C05461=1054.323,-117.646,435.270,170.401,28.686,155.440
C05462=1054.330,-117.397,435.261,170.403,28.687,155.440
C05463=1054.336,-117.147,435.251,170.405,28.688,155.440
C05464=1054.342,-116.897,435.242,170.407,28.688,155.440
C05465=1054.348,-116.647,435.232,170.409,28.689,155.440
C05466=1054.354,-116.397,435.222,170.410,28.689,155.440
C05467=1054.360,-116.148,435.213,170.412,28.689,155.440
C05468=1054.367,-115.898,435.203,170.415,28.691,155.440
C05469=1054.373,-115.648,435.194,170.417,28.691,155.440
C05470=1054.379,-115.364,435.183,170.419,28.692,155.440
C05471=1054.387,-115.080,435.172,170.422,28.692,155.440
C05472=1054.393,-114.795,435.162,170.424,28.693,155.440
C05473=1054.401,-114.511,435.150,170.427,28.694,155.439
C05474=1054.407,-114.261,435.141,170.428,28.694,155.439
C05475=1054.413,-114.011,435.131,170.430,28.695,155.439
C05476=1054.419,-113.762,435.122,170.432,28.696,155.439
C05477=1054.425,-113.512,435.113,170.434,28.696,155.439
C05478=1054.431,-113.263,435.103,170.436,28.697,155.439
C05479=1054.437,-113.013,435.092,170.439,28.698,155.439
C05480=1054.443,-112.763,435.083,170.441,28.698,155.439
C05481=1054.449,-112.514,435.073,170.443,28.699,155.439
C05482=1054.455,-112.264,435.063,170.445,28.699,155.439
C05483=1054.462,-112.014,435.054,170.446,28.700,155.439
C05484=1054.468,-111.764,435.044,170.448,28.701,155.439
C05485=1054.474,-111.514,435.035,170.450,28.702,155.439
C05486=1054.480,-111.265,435.025,170.453,28.702,155.439
C05487=1054.487,-111.015,435.015,170.455,28.703,155.439
C05488=1054.493,-110.766,435.005,170.457,28.704,155.439
C05489=1054.498,-110.515,434.995,170.459,28.704,155.439
C05490=1054.504,-110.266,434.986,170.461,28.705,155.439
C05491=1054.511,-110.016,434.976,170.462,28.706,155.439
C05492=1054.517,-109.766,434.966,170.465,28.706,155.438
C05493=1054.523,-109.517,434.956,170.467,28.707,155.438
C05494=1054.529,-109.267,434.947,170.469,28.708,155.438
C05495=1054.535,-109.017,434.937,170.471,28.708,155.438
C05496=1054.542,-108.768,434.927,170.473,28.709,155.438
C05497=1054.548,-108.518,434.917,170.475,28.710,155.438
C05498=1054.554,-108.268,434.907,170.477,28.711,155.438
C05499=1054.560,-108.018,434.897,170.479,28.711,155.438
C05500=1054.567,-107.768,434.888,170.481,28.712,155.438
C05501=1054.573,-107.519,434.877,170.483,28.713,155.438
C05502=1054.579,-107.269,434.868,170.485,28.713,155.438
C05503=1054.585,-107.019,434.858,170.487,28.714,155.438
C05504=1054.591,-106.769,434.848,170.489,28.715,155.438
C05505=1054.597,-106.520,434.838,170.491,28.716,155.438
C05506=1054.603,-106.270,434.828,170.494,28.716,155.438
C05507=1054.610,-106.020,434.819,170.495,28.717,155.438
C05508=1054.615,-105.771,434.808,170.497,28.719,155.438
C05509=1054.622,-105.521,434.798,170.499,28.719,155.438
C05510=1054.628,-105.271,434.789,170.501,28.720,155.438
C05511=1054.634,-105.022,434.778,170.503,28.720,155.438
C05512=1054.640,-104.772,434.768,170.505,28.721,155.438
C05513=1054.646,-104.521,434.758,170.508,28.722,155.438
C05514=1054.653,-104.272,434.748,170.509,28.723,155.438
C05515=1054.658,-104.022,434.738,170.511,28.724,155.438
C05516=1054.665,-103.773,434.727,170.513,28.725,155.438
C05517=1054.671,-103.523,434.718,170.515,28.726,155.438
C05518=1054.677,-103.273,434.708,170.517,28.726,155.438
C05519=1054.683,-103.024,434.697,170.519,28.727,155.438
C05520=1054.689,-102.774,434.688,170.522,28.728,155.438
C05521=1054.695,-102.525,434.678,170.523,28.729,155.438
C05522=1054.702,-102.274,434.667,170.525,28.730,155.438
C05523=1054.708,-102.025,434.657,170.527,28.731,155.438
C05524=1054.714,-101.775,434.647,170.529,28.731,155.438
C05525=1054.720,-101.525,434.637,170.531,28.732,155.438
C05526=1054.726,-101.276,434.627,170.533,28.733,155.438
C05527=1054.732,-101.026,434.617,170.536,28.734,155.437
C05528=1054.738,-100.777,434.606,170.537,28.735,155.438
C05529=1054.745,-100.526,434.596,170.539,28.736,155.438
C05530=1054.751,-100.277,434.586,170.541,28.737,155.437
C05531=1054.757,-100.027,434.576,170.543,28.738,155.437
C05532=1054.763,-99.778,434.566,170.545,28.739,155.438
C05533=1054.769,-99.527,434.555,170.547,28.739,155.437
C05534=1054.777,-99.242,434.544,170.550,28.740,155.437
C05535=1054.784,-98.956,434.532,170.551,28.741,155.437
C05536=1054.791,-98.670,434.521,170.554,28.743,155.437
C05537=1054.798,-98.385,434.508,170.556,28.744,155.437
C05538=1054.803,-98.135,434.498,170.558,28.744,155.437
C05539=1054.810,-97.886,434.488,170.560,28.745,155.437
C05540=1054.816,-97.636,434.478,170.563,28.746,155.437
C05541=1054.822,-97.386,434.467,170.564,28.747,155.437
C05542=1054.829,-97.137,434.457,170.566,28.748,155.437
C05543=1054.834,-96.887,434.447,170.568,28.749,155.437
C05544=1054.840,-96.637,434.436,170.570,28.750,155.437
C05545=1054.847,-96.388,434.425,170.572,28.751,155.437
C05546=1054.852,-96.138,434.415,170.574,28.752,155.438
C05547=1054.859,-95.888,434.405,170.575,28.753,155.438
C05548=1054.865,-95.638,434.394,170.578,28.754,155.438
C05549=1054.871,-95.389,434.384,170.580,28.755,155.438
C05550=1054.877,-95.139,434.373,170.582,28.756,155.438
C05551=1054.882,-94.890,434.362,170.584,28.757,155.438
C05552=1054.889,-94.639,434.352,170.586,28.758,155.438
C05553=1054.895,-94.390,434.342,170.587,28.759,155.438
C05554=1054.901,-94.140,434.331,170.589,28.760,155.438
C05555=1054.907,-93.890,434.321,170.591,28.761,155.438
C05556=1054.913,-93.641,434.310,170.594,28.763,155.438
C05557=1054.920,-93.391,434.300,170.596,28.763,155.438
C05558=1054.925,-93.141,434.289,170.598,28.764,155.438
C05559=1054.932,-92.892,434.279,170.600,28.765,155.438
C05560=1054.937,-92.642,434.268,170.601,28.766,155.438
C05561=1054.944,-92.392,434.257,170.603,28.767,155.438
C05562=1054.950,-92.143,434.247,170.605,28.768,155.438
C05563=1054.956,-91.893,434.237,170.607,28.769,155.438
C05564=1054.961,-91.643,434.226,170.610,28.771,155.438
C05565=1054.968,-91.393,434.215,170.611,28.772,155.438
C05566=1054.974,-91.144,434.204,170.613,28.773,155.438
C05567=1054.981,-90.895,434.194,170.615,28.774,155.438
C05568=1054.987,-90.644,434.183,170.617,28.775,155.438
C05569=1054.992,-90.394,434.173,170.619,28.776,155.438
C05570=1054.999,-90.145,434.162,170.621,28.777,155.438
C05571=1055.005,-89.895,434.151,170.622,28.778,155.438
C05572=1055.011,-89.645,434.140,170.624,28.780,155.438
C05573=1055.017,-89.396,434.130,170.627,28.781,155.438
C05574=1055.024,-89.146,434.119,170.629,28.782,155.438
C05575=1055.029,-88.896,434.108,170.631,28.783,155.438
C05576=1055.036,-88.647,434.098,170.633,28.784,155.438
C05577=1055.041,-88.397,434.087,170.634,28.785,155.438
C05578=1055.048,-88.147,434.076,170.636,28.786,155.438
C05579=1055.054,-87.898,434.066,170.638,28.787,155.438
C05580=1055.061,-87.648,434.055,170.640,28.788,155.438
C05581=1055.066,-87.398,434.044,170.643,28.789,155.438
C05582=1055.073,-87.149,434.033,170.645,28.790,155.438
C05583=1055.079,-86.899,434.022,170.646,28.791,155.439
C05584=1055.085,-86.649,434.011,170.648,28.792,155.439
C05585=1055.091,-86.400,434.001,170.650,28.794,155.439
C05586=1055.098,-86.150,433.990,170.652,28.795,155.439
C05587=1055.103,-85.901,433.979,170.654,28.796,155.439
C05588=1055.111,-85.651,433.968,170.656,28.797,155.439
C05589=1055.116,-85.401,433.957,170.657,28.798,155.439
C05590=1055.122,-85.152,433.946,170.660,28.799,155.439
C05591=1055.129,-84.902,433.936,170.662,28.800,155.439
C05592=1055.135,-84.652,433.925,170.664,28.801,155.439
C05593=1055.141,-84.402,433.914,170.666,28.803,155.439
C05594=1055.147,-84.153,433.903,170.667,28.804,155.439
C05595=1055.153,-83.903,433.892,170.669,28.805,155.439
C05596=1055.160,-83.653,433.881,170.671,28.806,155.439
C05597=1055.165,-83.404,433.870,170.673,28.807,155.439
C05598=1055.173,-83.120,433.858,170.676,28.808,155.439
C05599=1055.180,-82.837,433.846,170.678,28.810,155.439
C05600=1055.187,-82.553,433.833,170.680,28.811,155.439
C05601=1055.194,-82.270,433.821,170.682,28.812,155.439
C05602=1055.201,-82.020,433.810,170.684,28.814,155.439
C05603=1055.206,-81.771,433.799,170.686,28.815,155.440
C05604=1055.213,-81.521,433.788,170.688,28.816,155.440
C05605=1055.219,-81.271,433.777,170.689,28.817,155.440
C05606=1055.225,-81.021,433.766,170.691,28.818,155.440
C05607=1055.231,-80.772,433.755,170.694,28.820,155.440
C05608=1055.238,-80.522,433.745,170.696,28.821,155.440
C05609=1055.244,-80.273,433.733,170.698,28.822,155.440
C05610=1055.251,-80.023,433.722,170.700,28.823,155.440
C05611=1055.256,-79.773,433.711,170.701,28.825,155.440
C05612=1055.263,-79.523,433.700,170.703,28.826,155.440
C05613=1055.269,-79.274,433.689,170.705,28.827,155.440
C05614=1055.276,-79.024,433.678,170.707,28.828,155.440
C05615=1055.282,-78.775,433.666,170.709,28.829,155.440
C05616=1055.288,-78.525,433.655,170.710,28.830,155.440
C05617=1055.294,-78.275,433.644,170.713,28.832,155.440
C05618=1055.300,-78.025,433.633,170.715,28.833,155.440
C05619=1055.306,-77.776,433.622,170.717,28.835,155.441
C05620=1055.312,-77.526,433.610,170.719,28.836,155.441
C05621=1055.318,-77.276,433.599,170.720,28.837,155.441
C05622=1055.324,-77.026,433.588,170.722,28.839,155.441
C05623=1055.331,-76.777,433.577,170.724,28.840,155.441
C05624=1055.337,-76.527,433.565,170.726,28.841,155.441
C05625=1055.343,-76.278,433.554,170.728,28.842,155.441
C05626=1055.349,-76.027,433.543,170.730,28.843,155.441
C05627=1055.355,-75.779,433.532,170.731,28.845,155.441
C05628=1055.361,-75.528,433.520,170.734,28.846,155.441
C05629=1055.367,-75.279,433.509,170.736,28.848,155.441
C05630=1055.374,-75.029,433.498,170.738,28.849,155.441
C05631=1055.379,-74.780,433.487,170.739,28.851,155.441
C05632=1055.386,-74.530,433.475,170.741,28.852,155.442
C05633=1055.392,-74.281,433.464,170.743,28.853,155.442
C05634=1055.398,-74.031,433.453,170.745,28.854,155.442
C05635=1055.405,-73.780,433.441,170.747,28.856,155.442
C05636=1055.411,-73.532,433.430,170.749,28.857,155.442
C05637=1055.417,-73.281,433.418,170.750,28.859,155.442
C05638=1055.422,-73.032,433.406,170.752,28.860,155.442
C05639=1055.429,-72.782,433.395,170.754,28.861,155.442
C05640=1055.435,-72.533,433.383,170.757,28.863,155.442
C05641=1055.441,-72.283,433.372,170.758,28.864,155.442
C05642=1055.447,-72.033,433.361,170.760,28.866,155.442
C05643=1055.453,-71.784,433.349,170.762,28.867,155.443
C05644=1055.458,-71.534,433.338,170.764,28.868,155.443
C05645=1055.465,-71.284,433.326,170.766,28.870,155.443
C05646=1055.471,-71.035,433.315,170.767,28.872,155.443
C05647=1055.477,-70.785,433.303,170.769,28.873,155.443
C05648=1055.482,-70.536,433.292,170.771,28.874,155.443
C05649=1055.489,-70.286,433.280,170.773,28.876,155.443
C05650=1055.495,-70.036,433.268,170.775,28.877,155.443
C05651=1055.501,-69.787,433.256,170.776,28.879,155.443
C05652=1055.507,-69.536,433.245,170.778,28.880,155.444
C05653=1055.513,-69.288,433.233,170.780,28.881,155.444
C05654=1055.519,-69.037,433.222,170.783,28.883,155.444
C05655=1055.525,-68.788,433.210,170.784,28.885,155.444
C05656=1055.531,-68.538,433.199,170.786,28.886,155.444
C05657=1055.538,-68.288,433.187,170.788,28.887,155.444
C05658=1055.544,-68.040,433.175,170.790,28.889,155.444
C05659=1055.549,-67.789,433.163,170.792,28.891,155.444
C05660=1055.556,-67.540,433.151,170.793,28.892,155.444
C05661=1055.562,-67.290,433.141,170.795,28.893,155.445
C05662=1055.568,-67.009,433.127,170.797,28.895,155.445
C05663=1055.576,-66.728,433.114,170.800,28.897,155.445
C05664=1055.583,-66.446,433.100,170.801,28.898,155.445
C05665=1055.590,-66.165,433.087,170.803,28.900,155.445
C05666=1055.595,-65.915,433.076,170.805,28.902,155.445
C05667=1055.602,-65.666,433.064,170.807,28.903,155.445
C05668=1055.608,-65.416,433.052,170.809,28.904,155.445
C05669=1055.614,-65.167,433.041,170.810,28.906,155.446
C05670=1055.620,-64.917,433.028,170.813,28.908,155.446
C05671=1055.626,-64.667,433.016,170.815,28.909,155.446
C05672=1055.632,-64.418,433.006,170.817,28.911,155.446
C05673=1055.638,-64.168,432.993,170.819,28.912,155.446
C05674=1055.645,-63.918,432.981,170.820,28.914,155.446
C05675=1055.651,-63.669,432.970,170.822,28.915,155.446
C05676=1055.656,-63.419,432.958,170.824,28.916,155.446
C05677=1055.663,-63.169,432.946,170.826,28.918,155.447
C05678=1055.670,-62.920,432.934,170.827,28.920,155.447
C05679=1055.675,-62.670,432.922,170.829,28.921,155.447
C05680=1055.681,-62.421,432.910,170.831,28.922,155.447
C05681=1055.688,-62.171,432.898,170.833,28.924,155.447
C05682=1055.694,-61.921,432.886,170.835,28.926,155.447
C05683=1055.700,-61.672,432.875,170.836,28.927,155.447
C05684=1055.706,-61.422,432.863,170.838,28.929,155.448
C05685=1055.713,-61.172,432.851,170.840,28.930,155.448
C05686=1055.719,-60.923,432.838,170.842,28.932,155.448
C05687=1055.725,-60.674,432.827,170.844,28.933,155.448
C05688=1055.730,-60.423,432.815,170.845,28.935,155.448
C05689=1055.737,-60.174,432.803,170.848,28.937,155.448
C05690=1055.744,-59.924,432.791,170.850,28.938,155.448
C05691=1055.749,-59.675,432.779,170.852,28.939,155.448
C05692=1055.756,-59.425,432.767,170.853,28.941,155.448
C05693=1055.762,-59.175,432.756,170.855,28.943,155.449
C05694=1055.768,-58.925,432.743,170.857,28.944,155.449
C05695=1055.775,-58.676,432.731,170.859,28.946,155.449
C05696=1055.781,-58.427,432.720,170.861,28.947,155.449
C05697=1055.787,-58.177,432.707,170.862,28.949,155.449
C05698=1055.793,-57.927,432.695,170.864,28.950,155.449
C05699=1055.800,-57.678,432.683,170.866,28.952,155.449
C05700=1055.806,-57.428,432.671,170.868,28.953,155.450
C05701=1055.812,-57.179,432.659,170.869,28.955,155.450
C05702=1055.817,-56.928,432.647,170.871,28.957,155.450
C05703=1055.824,-56.679,432.635,170.873,28.958,155.450
C05704=1055.831,-56.429,432.623,170.875,28.960,155.450
C05705=1055.837,-56.179,432.611,170.877,28.961,155.450
C05706=1055.843,-55.930,432.599,170.878,28.962,155.450
C05707=1055.850,-55.680,432.587,170.880,28.964,155.450
C05708=1055.855,-55.431,432.575,170.882,28.966,155.451
C05709=1055.862,-55.182,432.563,170.884,28.967,155.451
C05710=1055.868,-54.932,432.550,170.885,28.969,155.451
C05711=1055.874,-54.682,432.538,170.887,28.971,155.451
C05712=1055.881,-54.433,432.526,170.890,28.972,155.451
C05713=1055.887,-54.183,432.514,170.892,28.974,155.451
C05714=1055.894,-53.933,432.502,170.894,28.976,155.451
C05715=1055.900,-53.683,432.489,170.895,28.977,155.452
C05716=1055.906,-53.434,432.477,170.897,28.979,155.452
C05717=1055.913,-53.184,432.465,170.899,28.981,155.452
C05718=1055.918,-52.935,432.453,170.901,28.982,155.452
C05719=1055.925,-52.685,432.441,170.902,28.983,155.452
C05720=1055.931,-52.435,432.428,170.904,28.985,155.452
C05721=1055.937,-52.186,432.416,170.906,28.986,155.452
C05722=1055.943,-51.936,432.404,170.908,28.988,155.453
C05723=1055.950,-51.686,432.392,170.910,28.990,155.453
C05724=1055.957,-51.437,432.379,170.911,28.991,155.453
C05725=1055.963,-51.188,432.367,170.913,28.993,155.453
C05726=1055.970,-50.907,432.353,170.915,28.995,155.453
C05727=1055.977,-50.628,432.339,170.918,28.997,155.453
C05728=1055.984,-50.347,432.325,170.919,28.999,155.454
C05729=1055.990,-50.067,432.312,170.921,29.000,155.454
C05730=1055.997,-49.818,432.299,170.923,29.002,155.454
C05731=1056.003,-49.569,432.286,170.925,29.004,155.454
C05732=1056.009,-49.319,432.274,170.926,29.006,155.454
C05733=1056.016,-49.069,432.262,170.928,29.007,155.454
C05734=1056.022,-48.819,432.249,170.930,29.009,155.455
C05735=1056.027,-48.571,432.236,170.932,29.011,155.455
C05736=1056.033,-48.321,432.224,170.933,29.013,155.455
C05737=1056.040,-48.071,432.212,170.935,29.014,155.455
C05738=1056.046,-47.821,432.199,170.937,29.016,155.455
C05739=1056.052,-47.571,432.187,170.939,29.018,155.455
C05740=1056.058,-47.322,432.174,170.941,29.019,155.456
C05741=1056.065,-47.073,432.162,170.942,29.021,155.456
C05742=1056.070,-46.823,432.149,170.944,29.023,155.456
C05743=1056.076,-46.573,432.137,170.946,29.025,155.456
C05744=1056.083,-46.324,432.123,170.948,29.026,155.456
C05745=1056.089,-46.074,432.111,170.949,29.028,155.456
C05746=1056.095,-45.824,432.099,170.951,29.030,155.457
C05747=1056.101,-45.575,432.085,170.953,29.032,155.457
C05748=1056.107,-45.325,432.073,170.955,29.033,155.457
C05749=1056.114,-45.075,432.061,170.956,29.035,155.457
C05750=1056.120,-44.826,432.048,170.958,29.037,155.457
C05751=1056.126,-44.576,432.035,170.960,29.039,155.458
C05752=1056.132,-44.326,432.023,170.962,29.041,155.458
C05753=1056.138,-44.077,432.009,170.963,29.042,155.458
C05754=1056.145,-43.828,431.997,170.965,29.044,155.458
C05755=1056.151,-43.578,431.985,170.967,29.046,155.458
C05756=1056.157,-43.328,431.972,170.969,29.048,155.458
C05757=1056.163,-43.078,431.959,170.970,29.049,155.459
C05758=1056.169,-42.829,431.946,170.972,29.051,155.459
C05759=1056.176,-42.580,431.934,170.974,29.053,155.459
C05760=1056.182,-42.330,431.921,170.976,29.055,155.459
C05761=1056.188,-42.081,431.908,170.978,29.056,155.459
C05762=1056.194,-41.831,431.895,170.979,29.058,155.460
C05763=1056.200,-41.581,431.883,170.981,29.060,155.460
C05764=1056.207,-41.332,431.870,170.983,29.062,155.460
C05765=1056.212,-41.082,431.858,170.984,29.064,155.460
C05766=1056.219,-40.833,431.844,170.986,29.066,155.460
C05767=1056.225,-40.583,431.832,170.988,29.067,155.461
C05768=1056.231,-40.334,431.819,170.990,29.069,155.461
C05769=1056.237,-40.084,431.807,170.992,29.071,155.461
C05770=1056.244,-39.835,431.793,170.993,29.073,155.461
C05771=1056.250,-39.584,431.780,170.995,29.074,155.461
C05772=1056.256,-39.335,431.767,170.997,29.076,155.462
C05773=1056.262,-39.085,431.755,170.999,29.078,155.462
C05774=1056.269,-38.836,431.741,171.000,29.080,155.462
C05775=1056.275,-38.586,431.729,171.002,29.082,155.462
C05776=1056.281,-38.337,431.716,171.004,29.084,155.462
C05777=1056.287,-38.087,431.703,171.006,29.085,155.462
C05778=1056.293,-37.837,431.690,171.007,29.087,155.463
C05779=1056.299,-37.587,431.677,171.009,29.089,155.463
C05780=1056.305,-37.338,431.664,171.011,29.091,155.463
C05781=1056.311,-37.089,431.651,171.013,29.093,155.463
C05782=1056.317,-36.839,431.638,171.014,29.095,155.463
C05783=1056.324,-36.589,431.624,171.016,29.097,155.464
C05784=1056.330,-36.339,431.612,171.018,29.099,155.464
C05785=1056.336,-36.090,431.599,171.020,29.100,155.464
C05786=1056.342,-35.841,431.585,171.021,29.103,155.464
C05787=1056.348,-35.591,431.573,171.023,29.104,155.464
C05788=1056.354,-35.342,431.559,171.025,29.106,155.465
C05789=1056.360,-35.092,431.547,171.026,29.108,155.465
C05790=1056.368,-34.812,431.531,171.028,29.110,155.465
C05791=1056.374,-34.533,431.517,171.030,29.112,155.465
C05792=1056.381,-34.253,431.503,171.032,29.114,155.466
C05793=1056.388,-33.974,431.487,171.033,29.116,155.466
C05794=1056.394,-33.724,431.475,171.035,29.119,155.466
C05795=1056.400,-33.475,431.461,171.037,29.120,155.466
C05796=1056.406,-33.226,431.448,171.039,29.122,155.467
C05797=1056.413,-32.975,431.435,171.040,29.124,155.467
C05798=1056.419,-32.726,431.422,171.042,29.126,155.467
C05799=1056.425,-32.477,431.409,171.044,29.128,155.467
C05800=1056.431,-32.227,431.395,171.046,29.130,155.467
C05801=1056.437,-31.977,431.383,171.047,29.132,155.468
C05802=1056.444,-31.728,431.369,171.049,29.134,155.468
C05803=1056.450,-31.478,431.356,171.051,29.135,155.468
C05804=1056.457,-31.229,431.343,171.053,29.138,155.468
C05805=1056.462,-30.979,431.329,171.054,29.139,155.468
C05806=1056.468,-30.729,431.316,171.056,29.142,155.469
C05807=1056.474,-30.480,431.303,171.058,29.143,155.469
C05808=1056.481,-30.230,431.289,171.060,29.145,155.469
C05809=1056.487,-29.980,431.277,171.061,29.147,155.469
C05810=1056.493,-29.731,431.263,171.063,29.149,155.470
C05811=1056.499,-29.482,431.250,171.064,29.151,155.470
C05812=1056.506,-29.232,431.236,171.066,29.153,155.470
C05813=1056.512,-28.983,431.223,171.068,29.154,155.470
C05814=1056.518,-28.733,431.209,171.069,29.157,155.470
C05815=1056.524,-28.483,431.197,171.071,29.158,155.471
C05816=1056.530,-28.234,431.183,171.073,29.160,155.471
C05817=1056.537,-27.984,431.170,171.075,29.162,155.471
C05818=1056.543,-27.735,431.157,171.076,29.164,155.471
C05819=1056.549,-27.485,431.143,171.078,29.166,155.472
C05820=1056.556,-27.235,431.130,171.080,29.168,155.472
C05821=1056.562,-26.986,431.116,171.081,29.170,155.472
C05822=1056.568,-26.737,431.103,171.083,29.172,155.472
C05823=1056.574,-26.487,431.089,171.085,29.174,155.472
C05824=1056.581,-26.237,431.076,171.087,29.176,155.473
C05825=1056.586,-25.987,431.062,171.088,29.178,155.473
C05826=1056.592,-25.738,431.049,171.090,29.180,155.473
C05827=1056.598,-25.489,431.036,171.092,29.182,155.473
C05828=1056.604,-25.238,431.022,171.093,29.184,155.474
C05829=1056.611,-24.989,431.008,171.094,29.186,155.474
C05830=1056.617,-24.740,430.995,171.096,29.188,155.474
C05831=1056.622,-24.490,430.981,171.098,29.190,155.474
C05832=1056.629,-24.240,430.968,171.100,29.192,155.474
C05833=1056.635,-23.991,430.954,171.101,29.194,155.475
C05834=1056.641,-23.741,430.941,171.103,29.196,155.475
C05835=1056.647,-23.492,430.927,171.105,29.198,155.475
C05836=1056.653,-23.242,430.913,171.107,29.200,155.475
C05837=1056.659,-22.993,430.900,171.108,29.202,155.476
C05838=1056.666,-22.744,430.886,171.110,29.205,155.476
C05839=1056.672,-22.494,430.872,171.112,29.206,155.476
C05840=1056.678,-22.244,430.858,171.114,29.208,155.476
C05841=1056.684,-21.995,430.845,171.115,29.211,155.477
C05842=1056.690,-21.745,430.831,171.116,29.212,155.477
C05843=1056.697,-21.496,430.818,171.118,29.214,155.477
C05844=1056.702,-21.246,430.804,171.120,29.216,155.477
C05845=1056.709,-20.996,430.790,171.121,29.219,155.478
C05846=1056.715,-20.747,430.777,171.123,29.220,155.478
C05847=1056.721,-20.497,430.763,171.125,29.222,155.478
C05848=1056.727,-20.247,430.749,171.126,29.225,155.478
C05849=1056.733,-19.998,430.735,171.128,29.227,155.479
C05850=1056.739,-19.749,430.721,171.130,29.228,155.479
C05851=1056.746,-19.499,430.708,171.132,29.231,155.479
C05852=1056.752,-19.249,430.694,171.133,29.233,155.479
C05853=1056.758,-19.000,430.681,171.135,29.235,155.480
C05854=1056.765,-18.720,430.664,171.137,29.237,155.480
C05855=1056.772,-18.440,430.649,171.139,29.239,155.480
C05856=1056.779,-18.159,430.634,171.140,29.242,155.480
C05857=1056.786,-17.879,430.618,171.142,29.244,155.481
C05858=1056.792,-17.630,430.604,171.144,29.246,155.481
C05859=1056.798,-17.380,430.591,171.146,29.248,155.481
C05860=1056.804,-17.130,430.577,171.147,29.250,155.481
C05861=1056.811,-16.881,430.563,171.149,29.252,155.482
C05862=1056.818,-16.631,430.549,171.151,29.254,155.482
C05863=1056.823,-16.382,430.535,171.153,29.256,155.482
C05864=1056.829,-16.133,430.522,171.153,29.258,155.482
C05865=1056.836,-15.883,430.507,171.155,29.260,155.483
C05866=1056.842,-15.634,430.494,171.157,29.262,155.483
C05867=1056.848,-15.383,430.480,171.158,29.264,155.483
C05868=1056.854,-15.134,430.466,171.160,29.266,155.483
C05869=1056.861,-14.884,430.451,171.162,29.268,155.484
C05870=1056.867,-14.635,430.438,171.164,29.270,155.484
C05871=1056.872,-14.386,430.424,171.165,29.273,155.484
C05872=1056.879,-14.136,430.409,171.167,29.275,155.484
C05873=1056.885,-13.887,430.396,171.169,29.277,155.485
C05874=1056.891,-13.636,430.382,171.170,29.279,155.485
C05875=1056.897,-13.388,430.368,171.171,29.281,155.485
C05876=1056.903,-13.138,430.354,171.173,29.283,155.486
C05877=1056.909,-12.889,430.339,171.175,29.285,155.486
C05878=1056.916,-12.639,430.326,171.177,29.287,155.486
C05879=1056.922,-12.389,430.312,171.178,29.289,155.486
C05880=1056.927,-12.140,430.297,171.180,29.292,155.487
C05881=1056.934,-11.890,430.283,171.182,29.294,155.487
C05882=1056.940,-11.641,430.269,171.184,29.296,155.487
C05883=1056.946,-11.391,430.254,171.184,29.298,155.487
C05884=1056.952,-11.142,430.241,171.186,29.300,155.488
C05885=1056.958,-10.893,430.227,171.188,29.302,155.488
C05886=1056.964,-10.642,430.212,171.189,29.305,155.488
C05887=1056.971,-10.394,430.198,171.191,29.307,155.488
C05888=1056.977,-10.143,430.184,171.193,29.309,155.489
C05889=1056.983,-9.894,430.170,171.195,29.311,155.489
C05890=1056.989,-9.644,430.156,171.196,29.313,155.489
C05891=1056.995,-9.396,430.141,171.197,29.315,155.489
C05892=1057.001,-9.145,430.127,171.199,29.317,155.490
C05893=1057.008,-8.897,430.113,171.201,29.319,155.490
C05894=1057.014,-8.646,430.099,171.202,29.321,155.490
C05895=1057.020,-8.397,430.084,171.204,29.324,155.491
C05896=1057.026,-8.147,430.070,171.206,29.326,155.491
C05897=1057.032,-7.898,430.056,171.208,29.328,155.491
C05898=1057.038,-7.648,430.042,171.209,29.330,155.491
C05899=1057.045,-7.399,430.027,171.210,29.332,155.492
C05900=1057.051,-7.149,430.014,171.212,29.334,155.492
C05901=1057.057,-6.900,429.999,171.214,29.337,155.492
C05902=1057.063,-6.650,429.985,171.215,29.339,155.493
C05903=1057.070,-6.401,429.971,171.217,29.341,155.493
C05904=1057.076,-6.152,429.956,171.219,29.343,155.493
C05905=1057.082,-5.901,429.942,171.220,29.345,155.493
C05906=1057.087,-5.652,429.927,171.222,29.348,155.494
C05907=1057.094,-5.403,429.914,171.223,29.350,155.494
C05908=1057.101,-5.153,429.899,171.225,29.352,155.494
C05909=1057.106,-4.904,429.884,171.226,29.353,155.494
C05910=1057.113,-4.654,429.870,171.228,29.356,155.495
C05911=1057.119,-4.405,429.856,171.230,29.358,155.495
C05912=1057.125,-4.155,429.841,171.232,29.360,155.495
C05913=1057.131,-3.905,429.827,171.233,29.362,155.495
C05914=1057.138,-3.656,429.813,171.235,29.364,155.496
C05915=1057.144,-3.407,429.798,171.236,29.366,155.496
C05916=1057.150,-3.157,429.784,171.238,29.368,155.496
C05917=1057.156,-2.908,429.769,171.239,29.371,155.497
C05918=1057.163,-2.625,429.752,171.241,29.373,155.497
C05919=1057.169,-2.344,429.736,171.243,29.376,155.497
C05920=1057.177,-2.062,429.720,171.244,29.378,155.498
C05921=1057.184,-1.780,429.703,171.246,29.381,155.498
C05922=1057.189,-1.531,429.688,171.248,29.383,155.498
C05923=1057.196,-1.281,429.674,171.250,29.386,155.499
C05924=1057.201,-1.032,429.660,171.251,29.388,155.499
C05925=1057.208,-0.782,429.645,171.253,29.390,155.499
C05926=1057.214,-0.532,429.630,171.255,29.392,155.499
C05927=1057.220,-0.284,429.615,171.256,29.395,155.500
C05928=1057.226,-0.033,429.601,171.257,29.397,155.500
C05929=1057.232,0.216,429.586,171.259,29.399,155.500
C05930=1057.238,0.465,429.571,171.261,29.401,155.501
C05931=1057.244,0.715,429.556,171.262,29.404,155.501
C05932=1057.250,0.964,429.542,171.264,29.406,155.501
C05933=1057.257,1.214,429.527,171.266,29.408,155.501
C05934=1057.262,1.463,429.513,171.267,29.410,155.502
C05935=1057.268,1.713,429.498,171.268,29.413,155.502
C05936=1057.274,1.963,429.483,171.270,29.415,155.502
C05937=1057.280,2.212,429.468,171.272,29.417,155.503
C05938=1057.286,2.461,429.453,171.274,29.419,155.503
C05939=1057.293,2.711,429.438,171.275,29.421,155.503
C05940=1057.298,2.960,429.424,171.276,29.423,155.504
C05941=1057.305,3.210,429.409,171.278,29.426,155.504
C05942=1057.311,3.460,429.394,171.279,29.428,155.504
C05943=1057.317,3.709,429.380,171.281,29.431,155.504
C05944=1057.323,3.959,429.365,171.283,29.433,155.505
C05945=1057.329,4.208,429.350,171.285,29.435,155.505
C05946=1057.335,4.457,429.335,171.285,29.437,155.505
C05947=1057.342,4.707,429.320,171.287,29.440,155.506
C05948=1057.348,4.957,429.305,171.289,29.442,155.506
C05949=1057.354,5.205,429.291,171.291,29.444,155.506
C05950=1057.360,5.455,429.276,171.292,29.446,155.507
C05951=1057.366,5.705,429.261,171.294,29.448,155.507
C05952=1057.372,5.954,429.246,171.295,29.450,155.507
C05953=1057.378,6.204,429.231,171.296,29.453,155.508
C05954=1057.384,6.453,429.216,171.298,29.455,155.508
C05955=1057.391,6.703,429.201,171.300,29.458,155.508
C05956=1057.396,6.952,429.186,171.302,29.460,155.508
C05957=1057.403,7.202,429.171,171.303,29.462,155.509
C05958=1057.409,7.451,429.156,171.304,29.464,155.509
C05959=1057.415,7.700,429.142,171.306,29.467,155.509
C05960=1057.421,7.950,429.127,171.308,29.469,155.510
C05961=1057.428,8.200,429.112,171.309,29.471,155.510
C05962=1057.434,8.449,429.097,171.311,29.473,155.510
C05963=1057.440,8.698,429.082,171.313,29.475,155.510
C05964=1057.446,8.948,429.067,171.314,29.477,155.511
C05965=1057.452,9.198,429.052,171.315,29.480,155.511
C05966=1057.459,9.447,429.036,171.317,29.482,155.511
C05967=1057.465,9.696,429.021,171.319,29.485,155.512
C05968=1057.471,9.945,429.007,171.321,29.487,155.512
C05969=1057.477,10.195,428.992,171.322,29.489,155.512
C05970=1057.484,10.445,428.977,171.323,29.491,155.513
C05971=1057.490,10.694,428.962,171.325,29.494,155.513
C05972=1057.495,10.944,428.947,171.326,29.496,155.513
C05973=1057.501,11.193,428.932,171.328,29.498,155.513
C05974=1057.508,11.442,428.916,171.330,29.500,155.514
C05975=1057.514,11.692,428.901,171.332,29.502,155.514
C05976=1057.521,11.942,428.886,171.332,29.504,155.514
C05977=1057.527,12.191,428.871,171.334,29.507,155.515
C05978=1057.533,12.440,428.857,171.336,29.509,155.515
C05979=1057.539,12.690,428.842,171.338,29.512,155.515
C05980=1057.545,12.939,428.826,171.339,29.514,155.516
C05981=1057.552,13.189,428.811,171.340,29.516,155.516
C05982=1057.559,13.472,428.794,171.342,29.518,155.516
C05983=1057.566,13.756,428.776,171.344,29.521,155.517
C05984=1057.573,14.041,428.759,171.346,29.524,155.517
C05985=1057.580,14.324,428.742,171.348,29.526,155.517
C05986=1057.587,14.573,428.727,171.350,29.529,155.518
C05987=1057.592,14.823,428.711,171.350,29.531,155.518
C05988=1057.599,15.073,428.696,171.352,29.533,155.518
C05989=1057.604,15.322,428.681,171.354,29.536,155.519
C05990=1057.610,15.571,428.666,171.356,29.538,155.519
C05991=1057.617,15.821,428.651,171.357,29.540,155.519
C05992=1057.623,16.070,428.634,171.358,29.542,155.519
C05993=1057.629,16.320,428.619,171.360,29.545,155.520
C05994=1057.636,16.570,428.604,171.361,29.547,155.520
C05995=1057.641,16.818,428.589,171.363,29.550,155.520
C05996=1057.647,17.068,428.574,171.365,29.552,155.521
C05997=1057.653,17.318,428.558,171.366,29.554,155.521
C05998=1057.660,17.567,428.542,171.367,29.556,155.521
C05999=1057.666,17.817,428.527,171.369,29.559,155.522
C06000=1057.672,18.067,428.512,171.371,29.561,155.522
C06001=1057.678,18.316,428.496,171.373,29.564,155.522
C06002=1057.684,18.565,428.482,171.373,29.566,155.523
C06003=1057.690,18.814,428.465,171.375,29.568,155.523
C06004=1057.697,19.064,428.451,171.377,29.571,155.523
C06005=1057.702,19.313,428.435,171.379,29.573,155.524
C06006=1057.709,19.563,428.419,171.380,29.575,155.524
C06007=1057.715,19.812,428.404,171.381,29.577,155.524
C06008=1057.721,20.062,428.388,171.383,29.580,155.525
C06009=1057.728,20.311,428.373,171.385,29.582,155.525
C06010=1057.734,20.561,428.357,171.386,29.585,155.525
C06011=1057.739,20.809,428.342,171.388,29.587,155.526
C06012=1057.745,21.059,428.326,171.389,29.589,155.526
C06013=1057.752,21.308,428.311,171.390,29.592,155.526
C06014=1057.758,21.558,428.295,171.392,29.594,155.527
C06015=1057.764,21.807,428.280,171.394,29.596,155.527
C06016=1057.770,22.057,428.264,171.395,29.598,155.527
C06017=1057.776,22.307,428.249,171.396,29.601,155.527
C06018=1057.782,22.556,428.232,171.398,29.603,155.528
C06019=1057.789,22.806,428.218,171.400,29.606,155.528
C06020=1057.795,23.055,428.201,171.402,29.608,155.528
C06021=1057.800,23.305,428.186,171.402,29.610,155.529
C06022=1057.807,23.554,428.170,171.404,29.612,155.529
C06023=1057.812,23.803,428.155,171.406,29.615,155.530
C06024=1057.819,24.052,428.139,171.408,29.617,155.530
C06025=1057.825,24.302,428.123,171.409,29.620,155.530
C06026=1057.831,24.551,428.108,171.410,29.622,155.531
C06027=1057.837,24.801,428.092,171.412,29.624,155.531
C06028=1057.843,25.050,428.077,171.413,29.626,155.531
C06029=1057.849,25.300,428.061,171.415,29.629,155.531
C06030=1057.856,25.549,428.045,171.416,29.631,155.532
C06031=1057.862,25.799,428.029,171.418,29.634,155.532
C06032=1057.868,26.048,428.013,171.419,29.636,155.532
C06033=1057.874,26.298,427.998,171.421,29.638,155.533
C06034=1057.880,26.547,427.982,171.423,29.641,155.533
C06035=1057.887,26.796,427.966,171.424,29.643,155.533
C06036=1057.892,27.046,427.951,171.425,29.646,155.534
C06037=1057.898,27.295,427.934,171.427,29.648,155.534
C06038=1057.905,27.544,427.919,171.429,29.650,155.534
C06039=1057.910,27.794,427.903,171.431,29.653,155.535
C06040=1057.917,28.043,427.888,171.431,29.655,155.535
C06041=1057.923,28.293,427.871,171.433,29.658,155.535
C06042=1057.929,28.542,427.855,171.435,29.660,155.536
C06043=1057.935,28.792,427.840,171.437,29.662,155.536
C06044=1057.941,29.041,427.824,171.437,29.665,155.536
C06045=1057.947,29.290,427.808,171.439,29.667,155.537
C06046=1057.954,29.576,427.789,171.441,29.669,155.537
C06047=1057.962,29.861,427.772,171.442,29.672,155.538
C06048=1057.968,30.145,427.753,171.444,29.675,155.538
C06049=1057.975,30.431,427.735,171.446,29.678,155.538
C06050=1057.981,30.680,427.718,171.447,29.681,155.539
C06051=1057.987,30.930,427.704,171.449,29.683,155.539
C06052=1057.993,31.179,427.687,171.451,29.685,155.539
C06053=1057.999,31.429,427.671,171.452,29.687,155.540
C06054=1058.005,31.678,427.655,171.453,29.690,155.540
C06055=1058.012,31.927,427.639,171.455,29.692,155.540
C06056=1058.018,32.176,427.623,171.457,29.695,155.541
C06057=1058.024,32.427,427.607,171.458,29.697,155.541
C06058=1058.030,32.676,427.591,171.459,29.700,155.541
C06059=1058.036,32.926,427.574,171.461,29.702,155.542
C06060=1058.043,33.175,427.559,171.463,29.704,155.542
C06061=1058.049,33.424,427.543,171.465,29.707,155.542
C06062=1058.055,33.673,427.526,171.465,29.709,155.543
C06063=1058.061,33.923,427.510,171.467,29.712,155.543
C06064=1058.066,34.172,427.494,171.469,29.714,155.543
C06065=1058.073,34.422,427.479,171.471,29.717,155.544
C06066=1058.079,34.671,427.463,171.471,29.719,155.544
C06067=1058.085,34.920,427.446,171.473,29.721,155.544
C06068=1058.091,35.170,427.430,171.475,29.723,155.545
C06069=1058.097,35.419,427.414,171.476,29.726,155.545
C06070=1058.104,35.669,427.398,171.478,29.728,155.545
C06071=1058.110,35.918,427.381,171.479,29.731,155.546
C06072=1058.116,36.168,427.365,171.481,29.733,155.546
C06073=1058.122,36.417,427.349,171.482,29.736,155.547
C06074=1058.128,36.666,427.333,171.484,29.738,155.547
C06075=1058.134,36.915,427.317,171.485,29.740,155.547
C06076=1058.140,37.165,427.301,171.487,29.743,155.548
C06077=1058.146,37.414,427.285,171.488,29.745,155.548
C06078=1058.153,37.664,427.268,171.490,29.748,155.548
C06079=1058.159,37.913,427.252,171.491,29.750,155.549
C06080=1058.165,38.163,427.235,171.493,29.752,155.549
C06081=1058.171,38.412,427.219,171.494,29.755,155.549
C06082=1058.177,38.661,427.203,171.496,29.757,155.550
C06083=1058.183,38.911,427.187,171.497,29.760,155.550
C06084=1058.189,39.160,427.170,171.499,29.762,155.550
C06085=1058.195,39.409,427.154,171.500,29.765,155.551
C06086=1058.201,39.660,427.138,171.502,29.767,155.551
C06087=1058.207,39.908,427.121,171.504,29.770,155.551
C06088=1058.213,40.158,427.104,171.505,29.772,155.552
C06089=1058.219,40.407,427.088,171.506,29.774,155.552
C06090=1058.225,40.656,427.072,171.508,29.777,155.552
C06091=1058.231,40.906,427.056,171.510,29.779,155.553
C06092=1058.237,41.155,427.039,171.510,29.782,155.553
C06093=1058.244,41.405,427.023,171.512,29.784,155.553
C06094=1058.250,41.654,427.006,171.514,29.787,155.554
C06095=1058.256,41.903,426.989,171.516,29.789,155.554
C06096=1058.262,42.152,426.973,171.516,29.792,155.555
C06097=1058.268,42.402,426.957,171.518,29.794,155.555
C06098=1058.274,42.651,426.941,171.520,29.796,155.555
C06099=1058.280,42.901,426.924,171.522,29.799,155.556
C06100=1058.286,43.151,426.908,171.522,29.801,155.556
C06101=1058.293,43.399,426.891,171.524,29.804,155.556
C06102=1058.299,43.693,426.871,171.526,29.807,155.557
C06103=1058.306,43.986,426.852,171.528,29.809,155.557
C06104=1058.313,44.279,426.833,171.529,29.813,155.558
C06105=1058.320,44.572,426.813,171.531,29.815,155.558
C06106=1058.326,44.817,426.796,171.533,29.818,155.558
C06107=1058.332,45.062,426.780,171.534,29.820,155.559
C06108=1058.337,45.308,426.764,171.536,29.823,155.559
C06109=1058.344,45.554,426.747,171.537,29.825,155.559
C06110=1058.349,45.799,426.731,171.539,29.828,155.560
C06111=1058.355,46.044,426.714,171.540,29.831,155.560
C06112=1058.361,46.289,426.697,171.541,29.833,155.561
C06113=1058.366,46.535,426.681,171.543,29.835,155.561
C06114=1058.372,46.784,426.665,171.545,29.838,155.561
C06115=1058.379,47.034,426.648,171.546,29.840,155.562
C06116=1058.384,47.283,426.631,171.547,29.843,155.562
C06117=1058.391,47.532,426.614,171.549,29.846,155.562
C06118=1058.397,47.782,426.598,171.551,29.848,155.563
C06119=1058.403,48.032,426.581,171.552,29.850,155.563
C06120=1058.409,48.281,426.563,171.553,29.853,155.564
C06121=1058.415,48.530,426.547,171.555,29.855,155.564
C06122=1058.421,48.779,426.531,171.556,29.858,155.564
C06123=1058.426,49.028,426.513,171.558,29.861,155.565
C06124=1058.433,49.278,426.497,171.559,29.863,155.565
C06125=1058.439,49.527,426.480,171.561,29.865,155.565
C06126=1058.445,49.776,426.464,171.562,29.868,155.566
C06127=1058.450,50.026,426.447,171.564,29.870,155.566
C06128=1058.457,50.276,426.429,171.565,29.873,155.566
C06129=1058.463,50.525,426.413,171.567,29.875,155.567
C06130=1058.469,50.774,426.395,171.568,29.878,155.567
C06131=1058.475,51.024,426.379,171.570,29.880,155.567
C06132=1058.481,51.273,426.362,171.571,29.882,155.568
C06133=1058.487,51.522,426.345,171.573,29.885,155.568
C06134=1058.493,51.771,426.328,171.574,29.888,155.569
C06135=1058.499,52.021,426.311,171.576,29.890,155.569
C06136=1058.505,52.270,426.294,171.577,29.893,155.569
C06137=1058.511,52.520,426.278,171.579,29.895,155.570
C06138=1058.518,52.769,426.260,171.580,29.897,155.570
C06139=1058.523,53.019,426.243,171.582,29.900,155.570
C06140=1058.529,53.267,426.226,171.583,29.903,155.571
C06141=1058.536,53.517,426.210,171.585,29.905,155.571
C06142=1058.541,53.766,426.192,171.586,29.908,155.571
C06143=1058.547,54.016,426.176,171.588,29.910,155.572
C06144=1058.554,54.265,426.159,171.589,29.912,155.572
C06145=1058.559,54.515,426.142,171.591,29.915,155.573
C06146=1058.565,54.764,426.125,171.592,29.917,155.573
C06147=1058.572,55.013,426.108,171.594,29.920,155.573
C06148=1058.578,55.263,426.091,171.595,29.923,155.574
C06149=1058.584,55.511,426.074,171.597,29.925,155.574
C06150=1058.590,55.762,426.057,171.598,29.927,155.574
C06151=1058.596,56.011,426.040,171.600,29.930,155.575
C06152=1058.602,56.259,426.023,171.601,29.932,155.575
C06153=1058.608,56.510,426.005,171.603,29.935,155.576
C06154=1058.614,56.758,425.988,171.604,29.937,155.576
C06155=1058.621,57.008,425.971,171.606,29.940,155.576
C06156=1058.626,57.257,425.954,171.607,29.942,155.577
C06157=1058.633,57.506,425.937,171.609,29.944,155.577
C06158=1058.639,57.756,425.921,171.610,29.947,155.577
C06159=1058.645,58.005,425.903,171.612,29.950,155.578
C06160=1058.651,58.255,425.886,171.613,29.952,155.578
C06161=1058.657,58.504,425.868,171.614,29.955,155.578
C06162=1058.663,58.753,425.852,171.616,29.957,155.579
C06163=1058.670,59.003,425.834,171.618,29.959,155.579
C06164=1058.675,59.252,425.817,171.619,29.962,155.580
C06165=1058.682,59.502,425.800,171.621,29.964,155.580
C06166=1058.687,59.751,425.783,171.622,29.967,155.580
C06167=1058.694,60.000,425.765,171.624,29.969,155.580
C06168=1058.700,60.249,425.748,171.625,29.972,155.581
C06169=1058.706,60.499,425.731,171.626,29.974,155.581
C06170=1058.713,60.748,425.714,171.628,29.976,155.582
C06171=1058.718,60.997,425.697,171.630,29.979,155.582
C06172=1058.725,61.246,425.679,171.631,29.981,155.582
C06173=1058.731,61.496,425.663,171.633,29.984,155.583
C06174=1058.738,61.781,425.642,171.634,29.987,155.583
C06175=1058.745,62.066,425.623,171.636,29.989,155.584
C06176=1058.752,62.351,425.603,171.638,29.992,155.584
C06177=1058.759,62.635,425.583,171.639,29.995,155.584
C06178=1058.766,62.885,425.567,171.641,29.998,155.585
C06179=1058.771,63.134,425.549,171.643,30.000,155.585
C06180=1058.778,63.383,425.532,171.644,30.002,155.585
C06181=1058.784,63.632,425.514,171.645,30.005,155.586
C06182=1058.791,63.882,425.497,171.647,30.007,155.586
C06183=1058.796,64.131,425.479,171.649,30.010,155.587
C06184=1058.803,64.380,425.462,171.651,30.012,155.587
C06185=1058.808,64.630,425.445,171.651,30.015,155.587
C06186=1058.815,64.879,425.428,171.653,30.017,155.588
C06187=1058.821,65.128,425.410,171.655,30.020,155.588
C06188=1058.827,65.378,425.392,171.656,30.022,155.588
C06189=1058.833,65.627,425.375,171.657,30.025,155.589
C06190=1058.839,65.876,425.358,171.659,30.027,155.589
C06191=1058.845,66.126,425.340,171.661,30.030,155.589
C06192=1058.851,66.374,425.323,171.662,30.032,155.590
C06193=1058.857,66.624,425.305,171.663,30.035,155.590
C06194=1058.863,66.873,425.287,171.665,30.038,155.591
C06195=1058.869,67.123,425.270,171.667,30.040,155.591
C06196=1058.876,67.372,425.252,171.668,30.042,155.591
C06197=1058.881,67.621,425.235,171.669,30.045,155.592
C06198=1058.887,67.871,425.217,171.671,30.047,155.592
C06199=1058.893,68.120,425.200,171.673,30.050,155.592
C06200=1058.900,68.370,425.182,171.674,30.052,155.593
C06201=1058.905,68.619,425.164,171.675,30.055,155.593
C06202=1058.912,68.868,425.147,171.677,30.057,155.594
C06203=1058.917,69.117,425.129,171.679,30.060,155.594
C06204=1058.924,69.367,425.111,171.680,30.063,155.594
C06205=1058.929,69.616,425.094,171.682,30.065,155.595
C06206=1058.936,69.865,425.076,171.683,30.067,155.595
C06207=1058.941,70.114,425.059,171.685,30.070,155.595
C06208=1058.948,70.364,425.041,171.686,30.073,155.596
C06209=1058.953,70.613,425.023,171.688,30.075,155.596
C06210=1058.960,70.862,425.005,171.689,30.078,155.597
C06211=1058.965,71.111,424.987,171.691,30.080,155.597
C06212=1058.972,71.361,424.970,171.692,30.083,155.597
C06213=1058.978,71.610,424.952,171.694,30.085,155.598
C06214=1058.984,71.859,424.934,171.695,30.088,155.598
C06215=1058.990,72.109,424.916,171.697,30.090,155.599
C06216=1058.995,72.358,424.899,171.698,30.093,155.599
C06217=1059.002,72.607,424.880,171.700,30.095,155.599
C06218=1059.007,72.856,424.863,171.701,30.098,155.600
C06219=1059.014,73.106,424.845,171.703,30.100,155.600
C06220=1059.020,73.356,424.827,171.704,30.103,155.600
C06221=1059.026,73.605,424.810,171.706,30.105,155.601
C06222=1059.032,73.854,424.791,171.707,30.108,155.601
C06223=1059.038,74.103,424.774,171.709,30.111,155.602
C06224=1059.044,74.353,424.756,171.710,30.113,155.602
C06225=1059.049,74.602,424.738,171.712,30.115,155.602
C06226=1059.055,74.851,424.720,171.713,30.118,155.603
C06227=1059.062,75.100,424.701,171.715,30.121,155.603
C06228=1059.067,75.349,424.684,171.717,30.123,155.603
C06229=1059.074,75.599,424.667,171.718,30.125,155.604
C06230=1059.080,75.849,424.649,171.719,30.128,155.604
C06231=1059.086,76.097,424.630,171.721,30.131,155.605
C06232=1059.092,76.347,424.612,171.723,30.134,155.605
C06233=1059.098,76.596,424.595,171.724,30.136,155.605
C06234=1059.104,76.845,424.576,171.725,30.138,155.606
C06235=1059.110,77.095,424.558,171.727,30.141,155.606
C06236=1059.116,77.344,424.541,171.729,30.144,155.607
C06237=1059.122,77.593,424.522,171.730,30.146,155.607
C06238=1059.129,77.877,424.502,171.731,30.149,155.607
C06239=1059.136,78.163,424.481,171.733,30.152,155.608
C06240=1059.143,78.447,424.461,171.735,30.154,155.608
C06241=1059.150,78.731,424.440,171.737,30.158,155.609
C06242=1059.156,78.981,424.422,171.738,30.160,155.609
C06243=1059.161,79.230,424.404,171.740,30.163,155.609
C06244=1059.168,79.479,424.386,171.742,30.165,155.610
C06245=1059.173,79.729,424.367,171.743,30.168,155.610
C06246=1059.179,79.978,424.349,171.744,30.171,155.611
C06247=1059.185,80.227,424.331,171.746,30.173,155.611
C06248=1059.191,80.477,424.313,171.748,30.175,155.611
C06249=1059.197,80.726,424.295,171.749,30.178,155.612
C06250=1059.203,80.975,424.277,171.750,30.181,155.612
C06251=1059.210,81.224,424.258,171.752,30.183,155.613
C06252=1059.214,81.474,424.240,171.754,30.186,155.613
C06253=1059.221,81.723,424.221,171.755,30.188,155.613
C06254=1059.227,81.973,424.203,171.756,30.191,155.614
C06255=1059.233,82.221,424.185,171.758,30.193,155.614
C06256=1059.239,82.471,424.167,171.760,30.196,155.614
C06257=1059.245,82.720,424.148,171.761,30.199,155.615
C06258=1059.250,82.969,424.130,171.762,30.201,155.615
C06259=1059.257,83.218,424.112,171.764,30.204,155.616
C06260=1059.263,83.468,424.094,171.766,30.206,155.616
C06261=1059.269,83.717,424.075,171.767,30.209,155.616
C06262=1059.275,83.966,424.058,171.768,30.211,155.617
C06263=1059.281,84.215,424.039,171.770,30.214,155.617
C06264=1059.286,84.465,424.021,171.772,30.216,155.618
C06265=1059.292,84.714,424.002,171.774,30.219,155.618
C06266=1059.299,84.963,423.983,171.775,30.222,155.618
C06267=1059.305,85.213,423.965,171.776,30.224,155.619
C06268=1059.311,85.461,423.947,171.778,30.227,155.619
C06269=1059.316,85.711,423.929,171.780,30.229,155.619
C06270=1059.322,85.960,423.910,171.781,30.232,155.620
C06271=1059.329,86.210,423.891,171.782,30.234,155.620
C06272=1059.334,86.459,423.874,171.784,30.237,155.621
C06273=1059.341,86.708,423.855,171.786,30.240,155.621
C06274=1059.347,86.957,423.836,171.787,30.242,155.621
C06275=1059.353,87.207,423.818,171.788,30.244,155.622
C06276=1059.359,87.456,423.799,171.790,30.247,155.622
C06277=1059.365,87.705,423.782,171.792,30.250,155.623
C06278=1059.371,87.954,423.763,171.793,30.252,155.623
C06279=1059.377,88.204,423.744,171.794,30.255,155.623
C06280=1059.383,88.453,423.725,171.796,30.257,155.624
C06281=1059.389,88.702,423.707,171.798,30.260,155.624
C06282=1059.395,88.951,423.689,171.800,30.262,155.624
C06283=1059.401,89.200,423.670,171.801,30.265,155.625
C06284=1059.407,89.450,423.652,171.802,30.267,155.625
C06285=1059.413,89.699,423.633,171.804,30.270,155.626
C06286=1059.420,89.948,423.615,171.806,30.273,155.626
C06287=1059.426,90.197,423.596,171.807,30.275,155.626
C06288=1059.431,90.447,423.578,171.808,30.277,155.627
C06289=1059.437,90.696,423.559,171.810,30.280,155.627
C06290=1059.444,90.945,423.540,171.812,30.283,155.628
C06291=1059.449,91.194,423.521,171.814,30.285,155.628
C06292=1059.455,91.443,423.504,171.814,30.287,155.628
C06293=1059.461,91.693,423.484,171.816,30.290,155.629
C06294=1059.467,91.942,423.466,171.818,30.293,155.629
C06295=1059.473,92.191,423.446,171.820,30.296,155.630
C06296=1059.479,92.441,423.428,171.821,30.298,155.630
C06297=1059.484,92.689,423.409,171.822,30.301,155.630
C06298=1059.490,92.939,423.391,171.824,30.303,155.631
C06299=1059.496,93.188,423.372,171.826,30.306,155.631
C06300=1059.503,93.438,423.353,171.828,30.308,155.631
C06301=1059.509,93.687,423.334,171.828,30.311,155.632
C06302=1059.515,93.971,423.313,171.830,30.314,155.632
C06303=1059.522,94.256,423.291,171.832,30.317,155.633
C06304=1059.529,94.540,423.270,171.834,30.320,155.633
C06305=1059.536,94.826,423.249,171.835,30.323,155.634
C06306=1059.542,95.075,423.230,171.837,30.326,155.634
C06307=1059.548,95.324,423.211,171.839,30.328,155.635
C06308=1059.553,95.573,423.192,171.841,30.330,155.635
C06309=1059.559,95.822,423.173,171.842,30.333,155.635
C06310=1059.566,96.071,423.155,171.843,30.336,155.636
C06311=1059.571,96.321,423.135,171.845,30.338,155.636
C06312=1059.578,96.570,423.117,171.847,30.341,155.637
C06313=1059.583,96.819,423.097,171.848,30.344,155.637
C06314=1059.590,97.068,423.079,171.849,30.346,155.637
C06315=1059.596,97.318,423.060,171.851,30.348,155.638
C06316=1059.601,97.566,423.041,171.853,30.351,155.638
C06317=1059.607,97.815,423.022,171.854,30.354,155.638
C06318=1059.613,98.065,423.003,171.856,30.356,155.639
C06319=1059.619,98.314,422.984,171.857,30.359,155.639
C06320=1059.625,98.563,422.965,171.859,30.361,155.640
C06321=1059.631,98.813,422.946,171.861,30.364,155.640
C06322=1059.637,99.062,422.927,171.862,30.366,155.640
C06323=1059.643,99.311,422.908,171.864,30.369,155.641
C06324=1059.649,99.561,422.889,171.865,30.372,155.641
C06325=1059.655,99.810,422.870,171.867,30.374,155.642
C06326=1059.661,100.059,422.850,171.868,30.377,155.642
C06327=1059.668,100.308,422.832,171.870,30.379,155.642
C06328=1059.674,100.557,422.813,171.872,30.382,155.643
C06329=1059.680,100.806,422.794,171.873,30.384,155.643
C06330=1059.686,101.056,422.775,171.875,30.387,155.644
C06331=1059.691,101.305,422.755,171.876,30.390,155.644
C06332=1059.696,101.554,422.737,171.878,30.392,155.644
C06333=1059.703,101.803,422.718,171.880,30.395,155.645
C06334=1059.709,102.052,422.698,171.881,30.397,155.645
C06335=1059.715,102.301,422.679,171.882,30.400,155.646
C06336=1059.720,102.551,422.659,171.884,30.403,155.646
C06337=1059.727,102.800,422.641,171.886,30.405,155.646
C06338=1059.732,103.049,422.622,171.888,30.408,155.647
C06339=1059.738,103.298,422.602,171.889,30.411,155.647
C06340=1059.744,103.547,422.582,171.890,30.413,155.648
C06341=1059.751,103.797,422.564,171.892,30.416,155.648
C06342=1059.756,104.046,422.545,171.894,30.419,155.648
C06343=1059.762,104.295,422.525,171.896,30.421,155.649
C06344=1059.768,104.544,422.505,171.896,30.423,155.649
C06345=1059.774,104.793,422.487,171.898,30.426,155.650
C06346=1059.780,105.043,422.467,171.900,30.429,155.650
C06347=1059.786,105.292,422.447,171.902,30.431,155.650
C06348=1059.792,105.541,422.428,171.903,30.434,155.651
C06349=1059.797,105.790,422.409,171.904,30.437,155.651
C06350=1059.804,106.040,422.390,171.906,30.439,155.652
C06351=1059.810,106.288,422.370,171.908,30.442,155.652
C06352=1059.815,106.538,422.351,171.910,30.445,155.652
C06353=1059.821,106.787,422.332,171.911,30.447,155.653
C06354=1059.827,107.036,422.312,171.912,30.449,155.653
C06355=1059.834,107.285,422.293,171.914,30.452,155.654
C06356=1059.839,107.535,422.274,171.916,30.455,155.654
C06357=1059.845,107.783,422.254,171.917,30.457,155.654
C06358=1059.851,108.033,422.235,171.919,30.460,155.655
C06359=1059.857,108.282,422.215,171.921,30.463,155.655
C06360=1059.863,108.531,422.196,171.922,30.465,155.656
C06361=1059.869,108.780,422.177,171.924,30.467,155.656
C06362=1059.875,109.029,422.157,171.925,30.470,155.656
C06363=1059.881,109.278,422.138,171.927,30.473,155.657
C06364=1059.887,109.527,422.118,171.929,30.475,155.657
C06365=1059.893,109.776,422.099,171.930,30.478,155.658
C06366=1059.899,110.062,422.077,171.932,30.481,155.658
C06367=1059.906,110.346,422.054,171.934,30.484,155.658
C06368=1059.913,110.631,422.032,171.936,30.487,155.659
C06369=1059.920,110.915,422.009,171.938,30.490,155.659
C06370=1059.927,111.165,421.991,171.939,30.492,155.660
C06371=1059.933,111.413,421.971,171.940,30.495,155.660
C06372=1059.938,111.663,421.951,171.942,30.497,155.661
C06373=1059.944,111.912,421.931,171.944,30.500,155.661
C06374=1059.950,112.161,421.912,171.946,30.503,155.661
C06375=1059.956,112.410,421.892,171.947,30.505,155.662
C06376=1059.962,112.659,421.873,171.949,30.508,155.662
C06377=1059.968,112.909,421.853,171.950,30.511,155.663
C06378=1059.974,113.158,421.833,171.952,30.513,155.663
C06379=1059.980,113.407,421.813,171.953,30.516,155.663
C06380=1059.986,113.656,421.794,171.955,30.518,155.664
C06381=1059.992,113.905,421.774,171.957,30.521,155.664
C06382=1059.998,114.154,421.754,171.959,30.523,155.665
C06383=1060.004,114.404,421.735,171.960,30.526,155.665
C06384=1060.009,114.653,421.714,171.961,30.529,155.665
C06385=1060.014,114.902,421.695,171.963,30.531,155.666
C06386=1060.020,115.151,421.675,171.965,30.534,155.666
C06387=1060.026,115.400,421.655,171.967,30.537,155.667
C06388=1060.033,115.650,421.636,171.968,30.539,155.667
C06389=1060.038,115.899,421.615,171.969,30.542,155.667
C06390=1060.044,116.148,421.595,171.971,30.545,155.668
C06391=1060.050,116.397,421.576,171.973,30.547,155.668
C06392=1060.056,116.646,421.556,171.975,30.551,155.669
C06393=1060.062,116.895,421.536,171.976,30.553,155.669
C06394=1060.067,117.144,421.515,171.978,30.556,155.670
C06395=1060.073,117.393,421.496,171.979,30.558,155.670
C06396=1060.079,117.642,421.476,171.981,30.561,155.670
C06397=1060.085,117.891,421.456,171.982,30.564,155.671
C06398=1060.090,118.141,421.436,171.984,30.567,155.671
C06399=1060.096,118.390,421.416,171.986,30.569,155.672
C06400=1060.102,118.639,421.396,171.988,30.572,155.672
C06401=1060.108,118.888,421.376,171.989,30.574,155.673
C06402=1060.114,119.137,421.356,171.990,30.576,155.673
C06403=1060.119,119.386,421.336,171.992,30.579,155.673
C06404=1060.125,119.635,421.316,171.994,30.582,155.674
C06405=1060.132,119.885,421.296,171.996,30.585,155.674
C06406=1060.138,120.134,421.276,171.998,30.587,155.674
C06407=1060.143,120.383,421.256,171.999,30.590,155.675
C06408=1060.149,120.632,421.236,172.000,30.592,155.675
C06409=1060.155,120.881,421.216,172.002,30.595,155.676
C06410=1060.161,121.130,421.196,172.004,30.598,155.676
C06411=1060.166,121.380,421.176,172.005,30.600,155.677
C06412=1060.172,121.628,421.156,172.007,30.603,155.677
C06413=1060.178,121.877,421.136,172.009,30.606,155.677
C06414=1060.184,122.127,421.116,172.011,30.608,155.678
C06415=1060.190,122.377,421.095,172.012,30.611,155.678
C06416=1060.196,122.625,421.076,172.013,30.614,155.679
C06417=1060.202,122.874,421.056,172.015,30.616,155.679
C06418=1060.208,123.123,421.036,172.017,30.619,155.679
C06419=1060.214,123.373,421.015,172.019,30.622,155.680
C06420=1060.220,123.622,420.995,172.021,30.624,155.680
C06421=1060.226,123.870,420.975,172.022,30.627,155.681
C06422=1060.231,124.120,420.954,172.024,30.630,155.681
C06423=1060.238,124.369,420.934,172.025,30.632,155.682
C06424=1060.244,124.618,420.914,172.027,30.635,155.682
C06425=1060.250,124.867,420.894,172.028,30.638,155.682
C06426=1060.255,125.116,420.873,172.030,30.640,155.683
C06427=1060.261,125.365,420.853,172.032,30.643,155.683
C06428=1060.267,125.614,420.833,172.034,30.646,155.684
C06429=1060.273,125.863,420.813,172.036,30.648,155.684
C06430=1060.280,126.148,420.790,172.037,30.651,155.684
C06431=1060.286,126.432,420.767,172.039,30.654,155.685
C06432=1060.293,126.717,420.744,172.041,30.657,155.685
C06433=1060.300,127.002,420.720,172.043,30.660,155.686
C06434=1060.306,127.251,420.700,172.045,30.662,155.686
C06435=1060.312,127.500,420.680,172.046,30.665,155.687
C06436=1060.318,127.749,420.660,172.048,30.668,155.687
C06437=1060.324,127.998,420.639,172.050,30.670,155.687
C06438=1060.330,128.247,420.619,172.052,30.673,155.688
C06439=1060.336,128.496,420.598,172.053,30.676,155.688
C06440=1060.342,128.745,420.578,172.055,30.678,155.689
C06441=1060.348,128.994,420.557,172.056,30.681,155.689
C06442=1060.354,129.244,420.537,172.058,30.684,155.689
C06443=1060.360,129.493,420.517,172.060,30.686,155.690
C06444=1060.366,129.742,420.497,172.061,30.688,155.690
C06445=1060.372,129.991,420.476,172.063,30.691,155.691
C06446=1060.378,130.240,420.456,172.065,30.694,155.691
C06447=1060.384,130.489,420.435,172.067,30.696,155.691
C06448=1060.390,130.738,420.415,172.069,30.699,155.692
C06449=1060.396,130.987,420.395,172.070,30.702,155.692
C06450=1060.402,131.237,420.374,172.072,30.704,155.693
C06451=1060.408,131.485,420.354,172.074,30.707,155.693
C06452=1060.414,131.734,420.333,172.075,30.709,155.694
C06453=1060.420,131.984,420.312,172.077,30.712,155.694
C06454=1060.426,132.233,420.292,172.078,30.715,155.694
C06455=1060.432,132.481,420.272,172.080,30.717,155.695
C06456=1060.438,132.731,420.250,172.082,30.720,155.695
C06457=1060.444,132.979,420.230,172.084,30.723,155.696
C06458=1060.450,133.229,420.209,172.086,30.725,155.696
C06459=1060.455,133.478,420.189,172.087,30.728,155.696
C06460=1060.461,133.727,420.168,172.089,30.731,155.697
C06461=1060.467,133.976,420.147,172.091,30.734,155.697
C06462=1060.473,134.225,420.127,172.093,30.736,155.698
C06463=1060.479,134.474,420.106,172.094,30.739,155.698
C06464=1060.484,134.724,420.085,172.095,30.741,155.699
C06465=1060.490,134.972,420.065,172.097,30.744,155.699
C06466=1060.497,135.222,420.043,172.099,30.747,155.699
C06467=1060.503,135.470,420.023,172.101,30.749,155.700
C06468=1060.508,135.720,420.003,172.102,30.752,155.700
C06469=1060.514,135.969,419.981,172.104,30.755,155.701
C06470=1060.520,136.218,419.961,172.106,30.757,155.701
C06471=1060.526,136.467,419.940,172.108,30.760,155.701
C06472=1060.531,136.716,419.919,172.110,30.763,155.702
C06473=1060.538,136.965,419.899,172.111,30.765,155.702
C06474=1060.544,137.214,419.877,172.113,30.768,155.703
C06475=1060.549,137.463,419.857,172.115,30.771,155.703
C06476=1060.556,137.712,419.836,172.117,30.773,155.703
C06477=1060.561,137.961,419.815,172.119,30.776,155.704
C06478=1060.567,138.210,419.794,172.119,30.779,155.704
C06479=1060.573,138.459,419.774,172.121,30.781,155.705
C06480=1060.579,138.708,419.752,172.123,30.784,155.705
C06481=1060.584,138.957,419.731,172.125,30.786,155.706
C06482=1060.591,139.207,419.710,172.127,30.789,155.706
C06483=1060.597,139.455,419.690,172.128,30.792,155.706
C06484=1060.603,139.705,419.668,172.130,30.794,155.707
C06485=1060.608,139.954,419.648,172.132,30.797,155.707
C06486=1060.614,140.203,419.626,172.134,30.800,155.708
C06487=1060.620,140.452,419.606,172.136,30.803,155.708
C06488=1060.626,140.700,419.585,172.137,30.806,155.709
C06489=1060.632,140.950,419.564,172.139,30.808,155.709
C06490=1060.637,141.199,419.543,172.141,30.811,155.709
C06491=1060.643,141.448,419.521,172.143,30.814,155.710
C06492=1060.649,141.697,419.500,172.145,30.816,155.710
C06493=1060.655,141.946,419.479,172.146,30.819,155.711
C06494=1060.661,142.230,419.455,172.148,30.822,155.711
C06495=1060.668,142.515,419.432,172.150,30.825,155.712
C06496=1060.675,142.800,419.407,172.152,30.828,155.712
C06497=1060.682,143.084,419.383,172.154,30.832,155.713
C06498=1060.688,143.332,419.362,172.156,30.834,155.713
C06499=1060.693,143.582,419.341,172.158,30.837,155.713
C06500=1060.699,143.830,419.320,172.159,30.839,155.714
C06501=1060.705,144.080,419.298,172.161,30.842,155.714
C06502=1060.711,144.328,419.277,172.162,30.845,155.715
C06503=1060.717,144.578,419.256,172.164,30.847,155.715
C06504=1060.723,144.827,419.234,172.166,30.850,155.716
C06505=1060.729,145.075,419.214,172.168,30.853,155.716
C06506=1060.735,145.325,419.193,172.170,30.855,155.716
C06507=1060.740,145.574,419.171,172.171,30.858,155.717
C06508=1060.747,145.823,419.150,172.173,30.861,155.717
C06509=1060.752,146.071,419.128,172.175,30.864,155.718
C06510=1060.758,146.321,419.108,172.177,30.867,155.718
C06511=1060.764,146.571,419.086,172.179,30.869,155.719
C06512=1060.770,146.819,419.065,172.180,30.872,155.719
C06513=1060.776,147.068,419.043,172.182,30.875,155.719
C06514=1060.781,147.317,419.022,172.184,30.877,155.720
C06515=1060.787,147.567,419.001,172.186,30.880,155.720
C06516=1060.793,147.816,418.979,172.188,30.883,155.721
C06517=1060.799,148.064,418.958,172.190,30.885,155.721
C06518=1060.805,148.313,418.936,172.191,30.888,155.721
C06519=1060.811,148.562,418.915,172.193,30.890,155.722
C06520=1060.817,148.811,418.893,172.195,30.893,155.722
C06521=1060.822,149.060,418.872,172.197,30.896,155.723
C06522=1060.828,149.310,418.851,172.199,30.899,155.723
C06523=1060.834,149.559,418.830,172.200,30.902,155.724
C06524=1060.840,149.807,418.808,172.202,30.904,155.724
C06525=1060.846,150.056,418.787,172.204,30.907,155.725
C06526=1060.852,150.305,418.765,172.206,30.910,155.725
C06527=1060.858,150.554,418.744,172.208,30.912,155.725
C06528=1060.864,150.803,418.722,172.209,30.916,155.726
C06529=1060.869,151.052,418.700,172.211,30.918,155.726
C06530=1060.875,151.301,418.679,172.213,30.921,155.727
C06531=1060.881,151.551,418.657,172.215,30.923,155.727
C06532=1060.887,151.799,418.636,172.217,30.926,155.728
C06533=1060.893,152.048,418.614,172.218,30.929,155.728
C06534=1060.899,152.297,418.593,172.220,30.931,155.728
C06535=1060.904,152.546,418.571,172.222,30.935,155.729
C06536=1060.910,152.795,418.549,172.224,30.937,155.729
C06537=1060.916,153.044,418.528,172.226,30.940,155.730
C06538=1060.922,153.293,418.506,172.227,30.943,155.730
C06539=1060.928,153.542,418.484,172.229,30.945,155.731
C06540=1060.934,153.791,418.463,172.231,30.948,155.731
C06541=1060.939,154.040,418.441,172.233,30.951,155.731
C06542=1060.945,154.290,418.419,172.235,30.954,155.732
C06543=1060.951,154.538,418.398,172.236,30.956,155.732
C06544=1060.957,154.787,418.376,172.239,30.959,155.733
C06545=1060.963,155.036,418.354,172.241,30.962,155.733
C06546=1060.969,155.285,418.332,172.243,30.965,155.734
C06547=1060.974,155.534,418.310,172.245,30.967,155.734
C06548=1060.980,155.783,418.289,172.246,30.970,155.735
C06549=1060.987,156.032,418.267,172.248,30.973,155.735
C06550=1060.991,156.281,418.245,172.250,30.976,155.735
C06551=1060.998,156.530,418.223,172.252,30.978,155.736
C06552=1061.004,156.779,418.201,172.254,30.981,155.736
C06553=1061.009,157.028,418.179,172.255,30.984,155.737
C06554=1061.015,157.277,418.158,172.257,30.987,155.737
C06555=1061.021,157.526,418.136,172.259,30.990,155.738
C06556=1061.028,157.775,418.114,172.261,30.992,155.738
C06557=1061.033,158.024,418.092,172.263,30.995,155.738
C06558=1061.040,158.308,418.067,172.264,30.998,155.739
C06559=1061.046,158.592,418.042,172.267,31.001,155.739
C06560=1061.053,158.877,418.017,172.269,31.005,155.740
C06561=1061.060,159.160,417.992,172.271,31.007,155.740
C06562=1061.065,159.409,417.970,172.274,31.011,155.741
C06563=1061.072,159.659,417.948,172.275,31.013,155.741
C06564=1061.078,159.907,417.926,172.277,31.016,155.742
C06565=1061.083,160.156,417.904,172.279,31.019,155.742
C06566=1061.089,160.405,417.882,172.281,31.021,155.743
C06567=1061.095,160.655,417.861,172.283,31.024,155.743
C06568=1061.100,160.903,417.838,172.284,31.027,155.744
C06569=1061.107,161.152,417.816,172.286,31.030,155.744
C06570=1061.112,161.401,417.793,172.288,31.032,155.744
C06571=1061.118,161.650,417.771,172.290,31.036,155.745
C06572=1061.123,161.899,417.750,172.292,31.038,155.745
C06573=1061.129,162.148,417.727,172.294,31.041,155.746
C06574=1061.134,162.397,417.705,172.295,31.044,155.746
C06575=1061.140,162.645,417.683,172.297,31.047,155.747
C06576=1061.146,162.895,417.661,172.299,31.049,155.747
C06577=1061.151,163.144,417.638,172.302,31.053,155.748
C06578=1061.158,163.393,417.616,172.304,31.055,155.748
C06579=1061.163,163.641,417.593,172.305,31.059,155.749
C06580=1061.168,163.890,417.571,172.307,31.061,155.749
C06581=1061.175,164.139,417.549,172.309,31.064,155.749
C06582=1061.180,164.389,417.527,172.311,31.067,155.750
C06583=1061.185,164.637,417.504,172.313,31.070,155.750
C06584=1061.191,164.886,417.482,172.314,31.072,155.751
C06585=1061.197,165.135,417.459,172.316,31.076,155.751
C06586=1061.203,165.384,417.437,172.318,31.078,155.752
C06587=1061.208,165.633,417.414,172.320,31.081,155.752
C06588=1061.214,165.881,417.392,172.322,31.084,155.753
C06589=1061.220,166.131,417.370,172.324,31.087,155.753
C06590=1061.225,166.380,417.347,172.326,31.090,155.754
C06591=1061.231,166.629,417.325,172.328,31.093,155.754
C06592=1061.237,166.878,417.302,172.330,31.095,155.754
C06593=1061.242,167.126,417.280,172.332,31.099,155.755
C06594=1061.248,167.375,417.258,172.334,31.101,155.755
C06595=1061.254,167.624,417.235,172.335,31.104,155.756
C06596=1061.260,167.873,417.213,172.337,31.107,155.756
C06597=1061.265,168.122,417.190,172.339,31.110,155.757
C06598=1061.271,168.371,417.167,172.341,31.113,155.757
C06599=1061.277,168.620,417.146,172.344,31.116,155.758
C06600=1061.282,168.869,417.123,172.345,31.118,155.758
C06601=1061.288,169.118,417.100,172.347,31.122,155.759
C06602=1061.294,169.366,417.077,172.349,31.124,155.759
C06603=1061.300,169.616,417.055,172.351,31.127,155.760
C06604=1061.306,169.865,417.033,172.353,31.130,155.760
C06605=1061.311,170.113,417.010,172.354,31.133,155.761
C06606=1061.317,170.362,416.987,172.356,31.135,155.761
C06607=1061.323,170.612,416.965,172.359,31.139,155.761
C06608=1061.329,170.860,416.942,172.361,31.141,155.762
C06609=1061.335,171.109,416.919,172.363,31.145,155.762
C06610=1061.340,171.358,416.897,172.365,31.147,155.763
C06611=1061.346,171.607,416.875,172.366,31.150,155.763
C06612=1061.352,171.856,416.852,172.368,31.153,155.764
C06613=1061.358,172.105,416.829,172.370,31.156,155.764
C06614=1061.363,172.353,416.806,172.373,31.158,155.765
C06615=1061.370,172.602,416.784,172.375,31.162,155.765
C06616=1061.375,172.851,416.761,172.376,31.164,155.766
C06617=1061.381,173.100,416.739,172.378,31.167,155.766
C06618=1061.387,173.349,416.716,172.380,31.170,155.767
C06619=1061.392,173.598,416.693,172.382,31.173,155.767
C06620=1061.399,173.847,416.670,172.385,31.176,155.767
C06621=1061.405,174.096,416.647,172.387,31.179,155.768
C06622=1061.411,174.379,416.621,172.388,31.182,155.768
C06623=1061.418,174.663,416.596,172.391,31.185,155.769
C06624=1061.424,174.947,416.569,172.393,31.189,155.769
C06625=1061.431,175.231,416.543,172.396,31.192,155.770
C06626=1061.437,175.480,416.521,172.398,31.195,155.770
C06627=1061.443,175.729,416.498,172.399,31.197,155.771
C06628=1061.449,175.978,416.475,172.401,31.200,155.771
C06629=1061.454,176.226,416.452,172.403,31.203,155.772
C06630=1061.460,176.475,416.429,172.406,31.206,155.772
C06631=1061.466,176.724,416.406,172.408,31.209,155.773
C06632=1061.472,176.973,416.384,172.409,31.212,155.773
C06633=1061.478,177.222,416.361,172.411,31.214,155.774
C06634=1061.484,177.471,416.338,172.413,31.217,155.774
C06635=1061.490,177.720,416.315,172.416,31.220,155.775
C06636=1061.495,177.968,416.292,172.418,31.223,155.775
C06637=1061.502,178.218,416.269,172.420,31.226,155.775
C06638=1061.508,178.467,416.246,172.421,31.229,155.776
C06639=1061.514,178.715,416.223,172.423,31.232,155.776
C06640=1061.520,178.964,416.200,172.426,31.235,155.777
C06641=1061.526,179.213,416.177,172.428,31.237,155.777
C06642=1061.531,179.462,416.154,172.430,31.240,155.778
C06643=1061.537,179.710,416.131,172.431,31.243,155.778
C06644=1061.543,179.959,416.108,172.433,31.246,155.779
C06645=1061.550,180.209,416.085,172.436,31.249,155.779
C06646=1061.556,180.458,416.062,172.438,31.252,155.780
C06647=1061.562,180.706,416.039,172.440,31.254,155.780
C06648=1061.567,180.955,416.016,172.442,31.257,155.781
C06649=1061.573,181.204,415.993,172.444,31.260,155.781
C06650=1061.579,181.453,415.970,172.446,31.263,155.781
C06651=1061.585,181.701,415.947,172.448,31.266,155.782
C06652=1061.591,181.951,415.924,172.450,31.269,155.782
C06653=1061.597,182.199,415.900,172.453,31.272,155.783
C06654=1061.603,182.448,415.878,172.455,31.275,155.783
C06655=1061.609,182.697,415.855,172.456,31.277,155.784
C06656=1061.615,182.946,415.832,172.458,31.280,155.784
C06657=1061.621,183.195,415.808,172.461,31.283,155.785
C06658=1061.627,183.444,415.785,172.463,31.286,155.785
C06659=1061.633,183.692,415.762,172.465,31.289,155.786
C06660=1061.639,183.941,415.738,172.467,31.292,155.786
C06661=1061.645,184.190,415.715,172.469,31.294,155.786
C06662=1061.651,184.439,415.692,172.471,31.298,155.787
C06663=1061.657,184.688,415.669,172.473,31.300,155.787
C06664=1061.663,184.936,415.645,172.475,31.303,155.788
C06665=1061.668,185.186,415.622,172.478,31.307,155.788
C06666=1061.674,185.434,415.598,172.479,31.309,155.789
C06667=1061.680,185.683,415.575,172.481,31.313,155.789
C06668=1061.685,185.932,415.551,172.483,31.316,155.790
C06669=1061.691,186.181,415.528,172.486,31.319,155.790
C06670=1061.696,186.430,415.504,172.488,31.322,155.791
C06671=1061.702,186.678,415.480,172.490,31.325,155.791
C06672=1061.708,186.927,415.457,172.491,31.328,155.792
C06673=1061.713,187.176,415.433,172.494,31.331,155.792
C06674=1061.719,187.425,415.410,172.496,31.334,155.793
C06675=1061.726,187.674,415.386,172.498,31.337,155.793
C06676=1061.731,187.923,415.363,172.500,31.340,155.794
C06677=1061.737,188.171,415.339,172.503,31.343,155.794
C06678=1061.742,188.420,415.315,172.504,31.346,155.795
C06679=1061.748,188.669,415.292,172.506,31.349,155.795
C06680=1061.754,188.917,415.268,172.508,31.352,155.796
C06681=1061.759,189.167,415.244,172.511,31.355,155.796
C06682=1061.765,189.415,415.221,172.513,31.358,155.797
C06683=1061.770,189.664,415.197,172.514,31.361,155.797
C06684=1061.776,189.913,415.173,172.517,31.364,155.798
C06685=1061.782,190.163,415.149,172.519,31.367,155.798
C06686=1061.789,190.445,415.123,172.521,31.371,155.799
C06687=1061.796,190.729,415.095,172.524,31.374,155.799
C06688=1061.801,191.012,415.068,172.526,31.378,155.800
C06689=1061.809,191.295,415.041,172.528,31.381,155.801
C06690=1061.814,191.544,415.018,172.531,31.384,155.801
C06691=1061.820,191.793,414.994,172.533,31.387,155.802
C06692=1061.825,192.041,414.970,172.535,31.390,155.802
C06693=1061.832,192.290,414.946,172.538,31.393,155.803
C06694=1061.838,192.539,414.923,172.539,31.396,155.803
C06695=1061.843,192.788,414.899,172.541,31.399,155.804
C06696=1061.849,193.036,414.875,172.543,31.402,155.804
C06697=1061.855,193.286,414.851,172.546,31.405,155.805
C06698=1061.861,193.534,414.827,172.548,31.408,155.805
C06699=1061.866,193.783,414.803,172.550,31.412,155.806
C06700=1061.873,194.032,414.779,172.552,31.414,155.806
C06701=1061.878,194.280,414.755,172.554,31.417,155.807
C06702=1061.884,194.529,414.732,172.556,31.421,155.807
C06703=1061.890,194.779,414.707,172.559,31.423,155.808
C06704=1061.896,195.027,414.684,172.561,31.427,155.808
C06705=1061.901,195.275,414.659,172.563,31.430,155.809
C06706=1061.908,195.524,414.635,172.565,31.433,155.809
C06707=1061.912,195.774,414.612,172.567,31.436,155.810
C06708=1061.919,196.023,414.588,172.569,31.439,155.810
C06709=1061.925,196.271,414.564,172.572,31.442,155.811
C06710=1061.930,196.519,414.540,172.574,31.445,155.811
C06711=1061.937,196.768,414.516,172.577,31.448,155.812
C06712=1061.942,197.017,414.492,172.578,31.451,155.812
C06713=1061.949,197.266,414.467,172.580,31.454,155.813
C06714=1061.954,197.515,414.443,172.583,31.457,155.813
C06715=1061.960,197.763,414.420,172.585,31.460,155.814
C06716=1061.966,198.012,414.395,172.587,31.464,155.814
C06717=1061.972,198.260,414.371,172.590,31.466,155.815
C06718=1061.978,198.510,414.347,172.591,31.470,155.815
C06719=1061.984,198.758,414.322,172.593,31.473,155.816
C06720=1061.990,199.007,414.298,172.596,31.475,155.816
C06721=1061.995,199.256,414.274,172.598,31.479,155.817
C06722=1062.001,199.504,414.250,172.601,31.482,155.817
C06723=1062.007,199.753,414.226,172.603,31.485,155.818
C06724=1062.013,200.002,414.202,172.604,31.488,155.818
C06725=1062.019,200.251,414.178,172.607,31.491,155.819
C06726=1062.025,200.499,414.154,172.609,31.494,155.819
C06727=1062.031,200.749,414.129,172.612,31.497,155.820
C06728=1062.037,200.997,414.106,172.614,31.500,155.820
C06729=1062.043,201.246,414.081,172.616,31.503,155.821
C06730=1062.049,201.494,414.057,172.618,31.507,155.821
C06731=1062.055,201.744,414.033,172.620,31.509,155.822
C06732=1062.060,201.992,414.008,172.623,31.513,155.822
C06733=1062.067,202.241,413.984,172.625,31.516,155.823
C06734=1062.073,202.489,413.959,172.627,31.519,155.823
C06735=1062.079,202.739,413.935,172.630,31.522,155.824
C06736=1062.084,202.987,413.911,172.631,31.525,155.824
C06737=1062.090,203.236,413.886,172.634,31.529,155.825
C06738=1062.096,203.485,413.862,172.636,31.531,155.825
C06739=1062.102,203.733,413.837,172.638,31.534,155.826
C06740=1062.107,203.982,413.813,172.641,31.538,155.826
C06741=1062.113,204.231,413.788,172.643,31.541,155.827
C06742=1062.119,204.480,413.764,172.645,31.544,155.827
C06743=1062.125,204.728,413.738,172.647,31.547,155.828
C06744=1062.131,204.977,413.715,172.649,31.551,155.829
C06745=1062.137,205.226,413.690,172.652,31.554,155.829
C06746=1062.142,205.474,413.665,172.654,31.557,155.830
C06747=1062.148,205.723,413.641,172.657,31.560,155.830
C06748=1062.153,205.972,413.616,172.658,31.564,155.831
C06749=1062.160,206.221,413.591,172.661,31.567,155.831
C06750=1062.185,207.269,413.488,172.833,31.649,155.839
C06751=1062.190,207.495,413.465,172.835,31.653,155.840
C06752=1062.196,207.722,413.442,172.836,31.656,155.840
C06753=1062.201,207.947,413.418,172.838,31.660,155.841
C06754=1062.207,208.173,413.395,172.840,31.664,155.842
C06755=1062.212,208.400,413.372,172.841,31.668,155.842
C06756=1062.218,208.626,413.348,172.843,31.671,155.843
C06757=1062.223,208.853,413.325,172.845,31.675,155.844
C06758=1062.229,209.079,413.302,172.847,31.679,155.844
C06759=1062.236,209.327,413.276,172.849,31.683,155.845
C06760=1062.241,209.576,413.250,172.851,31.687,155.846
C06761=1062.247,209.825,413.225,172.852,31.691,155.847
C06762=1062.253,210.074,413.200,172.855,31.695,155.847
C06763=1062.260,210.322,413.174,172.857,31.699,155.848
C06764=1062.266,210.570,413.149,172.859,31.703,155.849
C06765=1062.271,210.819,413.123,172.861,31.707,155.849
C06766=1062.277,211.067,413.097,172.863,31.711,155.850
C06767=1062.283,211.316,413.072,172.864,31.715,155.851
C06768=1062.289,211.565,413.046,172.866,31.719,155.852
C06769=1062.295,211.813,413.020,172.868,31.723,155.852
C06770=1062.302,212.062,412.995,172.871,31.728,155.853
C06771=1062.308,212.311,412.969,172.873,31.731,155.854
C06772=1062.314,212.559,412.942,172.875,31.736,155.855
C06773=1062.320,212.808,412.917,172.876,31.739,155.855
C06774=1062.326,213.057,412.891,172.878,31.744,155.856
C06775=1062.332,213.306,412.866,172.880,31.748,155.857
C06776=1062.338,213.554,412.839,172.883,31.752,155.858
C06777=1062.344,213.803,412.814,172.885,31.756,155.858
C06778=1062.351,214.051,412.788,172.887,31.760,155.859
C06779=1062.356,214.300,412.762,172.888,31.764,155.860
C06780=1062.362,214.548,412.737,172.890,31.768,155.860
C06781=1062.368,214.797,412.710,172.892,31.772,155.861
C06782=1062.374,215.045,412.685,172.894,31.776,155.862
C06783=1062.380,215.294,412.658,172.897,31.780,155.863
C06784=1062.386,215.542,412.633,172.899,31.784,155.863
C06785=1062.392,215.791,412.606,172.901,31.788,155.864
C06786=1062.398,216.039,412.581,172.902,31.792,155.865
C06787=1062.404,216.288,412.555,172.904,31.796,155.866
C06788=1062.410,216.537,412.529,172.906,31.800,155.866
C06789=1062.416,216.785,412.503,172.909,31.804,155.867
C06790=1062.423,217.034,412.476,172.911,31.808,155.868
C06791=1062.428,217.283,412.450,172.913,31.812,155.869
C06792=1062.435,217.531,412.424,172.914,31.816,155.869
C06793=1062.440,217.780,412.398,172.916,31.820,155.870
C06794=1062.447,218.028,412.372,172.919,31.825,155.871
C06795=1062.452,218.277,412.346,172.921,31.828,155.871
C06796=1062.459,218.525,412.320,172.923,31.832,155.872
C06797=1062.464,218.774,412.294,172.925,31.836,155.873
C06798=1062.471,219.023,412.268,172.927,31.840,155.874
C06799=1062.477,219.271,412.241,172.929,31.844,155.874
C06800=1062.484,219.519,412.215,172.931,31.848,155.875
C06801=1062.489,219.768,412.189,172.933,31.852,155.876
C06802=1062.495,220.016,412.163,172.935,31.856,155.877
C06803=1062.502,220.266,412.136,172.937,31.860,155.877
C06804=1062.508,220.514,412.111,172.940,31.864,155.878
C06805=1062.514,220.763,412.084,172.941,31.868,155.879
C06806=1062.520,221.011,412.058,172.943,31.872,155.879
C06807=1062.525,221.240,412.034,172.945,31.876,155.880
C06808=1062.531,221.468,412.010,172.947,31.879,155.881
C06809=1062.537,221.697,411.986,172.949,31.883,155.881
C06810=1062.543,221.926,411.961,172.951,31.887,155.882
C06811=1062.548,222.155,411.937,172.953,31.891,155.883
C06812=1062.553,222.383,411.912,172.955,31.894,155.883
C06813=1062.559,222.612,411.888,172.956,31.898,155.884
C06814=1062.564,222.841,411.864,172.958,31.902,155.885
C06815=1062.571,223.089,411.838,172.961,31.905,155.885
C06816=1062.576,223.337,411.811,172.963,31.910,155.886
C06817=1062.583,223.586,411.784,172.965,31.913,155.887
C06818=1062.588,223.835,411.758,172.967,31.918,155.888
C06819=1062.595,224.083,411.732,172.970,31.922,155.888
C06820=1062.601,224.332,411.706,172.971,31.926,155.889
C06821=1062.606,224.580,411.679,172.973,31.929,155.890
C06822=1062.613,224.829,411.652,172.975,31.933,155.891
C06823=1062.618,225.077,411.625,172.978,31.938,155.891
C06824=1062.625,225.325,411.599,172.980,31.941,155.892
C06825=1062.631,225.574,411.573,172.982,31.946,155.893
C06826=1062.637,225.823,411.546,172.984,31.949,155.893
C06827=1062.643,226.071,411.519,172.986,31.954,155.894
C06828=1062.649,226.320,411.492,172.988,31.957,155.895
C06829=1062.656,226.568,411.466,172.990,31.961,155.896
C06830=1062.661,226.817,411.440,172.992,31.965,155.896
C06831=1062.667,227.066,411.413,172.995,31.969,155.897
C06832=1062.673,227.315,411.386,172.997,31.973,155.898
C06833=1062.679,227.563,411.360,172.999,31.977,155.899
C06834=1062.686,227.811,411.333,173.002,31.981,155.899
C06835=1062.692,228.059,411.306,173.003,31.985,155.900
C06836=1062.698,228.308,411.279,173.005,31.989,155.901
C06837=1062.704,228.556,411.253,173.007,31.993,155.901
C06838=1062.710,228.805,411.226,173.010,31.997,155.902
C06839=1062.716,229.054,411.199,173.012,32.001,155.903
C06840=1062.723,229.302,411.173,173.014,32.005,155.904
C06841=1062.729,229.551,411.146,173.017,32.009,155.904
C06842=1062.735,229.799,411.119,173.019,32.012,155.905
C06843=1062.740,230.048,411.093,173.020,32.017,155.906
C06844=1062.747,230.297,411.066,173.022,32.020,155.906
C06845=1062.753,230.544,411.038,173.025,32.025,155.907
C06846=1062.759,230.793,411.012,173.027,32.028,155.908
C06847=1062.765,231.042,410.985,173.029,32.033,155.909
C06848=1062.771,231.290,410.958,173.032,32.036,155.909
C06849=1062.777,231.538,410.931,173.034,32.040,155.910
C06850=1062.783,231.787,410.904,173.036,32.044,155.911
C06851=1062.789,232.035,410.877,173.038,32.048,155.911
C06852=1062.795,232.284,410.850,173.040,32.052,155.912
C06853=1062.801,232.533,410.823,173.042,32.056,155.913
C06854=1062.807,232.781,410.795,173.045,32.060,155.914
C06855=1062.813,233.030,410.768,173.047,32.064,155.914
C06856=1062.819,233.278,410.742,173.049,32.068,155.915
C06857=1062.825,233.527,410.714,173.051,32.072,155.916
C06858=1062.831,233.775,410.687,173.054,32.076,155.917
C06859=1062.837,234.023,410.661,173.055,32.080,155.917
C06860=1062.844,234.272,410.633,173.057,32.084,155.918
C06861=1062.849,234.520,410.606,173.060,32.088,155.919
C06862=1062.855,234.769,410.578,173.062,32.092,155.919
C06863=1062.861,234.993,410.554,173.064,32.095,155.920
C06864=1062.866,235.218,410.529,173.066,32.099,155.921
C06865=1062.872,235.443,410.505,173.068,32.102,155.921
C06866=1062.877,235.668,410.480,173.071,32.106,155.922
C06867=1062.883,235.892,410.456,173.073,32.110,155.923
C06868=1062.888,236.117,410.431,173.074,32.113,155.923
C06869=1062.893,236.341,410.406,173.076,32.117,155.924
C06870=1062.899,236.567,410.381,173.078,32.120,155.925
C06871=1062.905,236.815,410.355,173.080,32.124,155.925
C06872=1062.911,237.064,410.326,173.083,32.128,155.926
C06873=1062.917,237.312,410.300,173.085,32.132,155.927
C06874=1062.924,237.561,410.272,173.087,32.136,155.928
C06875=1062.930,237.808,410.245,173.090,32.140,155.928
C06876=1062.936,238.057,410.218,173.092,32.144,155.929
C06877=1062.941,238.305,410.190,173.094,32.148,155.930
C06878=1062.948,238.555,410.163,173.096,32.152,155.930
C06879=1062.954,238.802,410.135,173.098,32.156,155.931
C06880=1062.960,239.051,410.108,173.101,32.160,155.932
C06881=1062.966,239.299,410.080,173.103,32.163,155.933
C06882=1062.972,239.548,410.053,173.105,32.168,155.933
C06883=1062.978,239.796,410.026,173.108,32.171,155.934
C06884=1062.985,240.045,409.998,173.110,32.175,155.935
C06885=1062.990,240.293,409.970,173.113,32.179,155.936
C06886=1062.996,240.542,409.943,173.115,32.183,155.936
C06887=1063.003,240.790,409.916,173.116,32.187,155.937
C06888=1063.008,241.038,409.888,173.119,32.191,155.938
C06889=1063.015,241.287,409.861,173.121,32.195,155.938
C06890=1063.021,241.535,409.833,173.124,32.199,155.939
C06891=1063.027,241.784,409.805,173.126,32.203,155.940
C06892=1063.033,242.032,409.777,173.128,32.206,155.940
C06893=1063.039,242.281,409.750,173.131,32.210,155.941
C06894=1063.045,242.529,409.722,173.133,32.215,155.942
C06895=1063.051,242.777,409.695,173.136,32.218,155.943
C06896=1063.057,243.026,409.666,173.137,32.223,155.943
C06897=1063.063,243.274,409.639,173.139,32.226,155.944
C06898=1063.069,243.523,409.611,173.142,32.230,155.945
C06899=1063.076,243.771,409.584,173.144,32.234,155.946
C06900=1063.081,244.019,409.556,173.147,32.238,155.946
C06901=1063.088,244.268,409.528,173.149,32.242,155.947
C06902=1063.093,244.516,409.500,173.151,32.246,155.948
C06903=1063.100,244.764,409.472,173.154,32.250,155.948
C06904=1063.106,245.013,409.444,173.156,32.254,155.949
C06905=1063.112,245.261,409.417,173.159,32.258,155.950
C06906=1063.118,245.510,409.388,173.161,32.262,155.951
C06907=1063.124,245.758,409.361,173.163,32.266,155.951
C06908=1063.130,246.006,409.333,173.165,32.269,155.952
C06909=1063.136,246.255,409.305,173.167,32.274,155.953
C06910=1063.142,246.503,409.277,173.170,32.277,155.953
C06911=1063.148,246.751,409.249,173.172,32.282,155.954
C06912=1063.154,247.000,409.220,173.175,32.285,155.955
C06913=1063.160,247.248,409.193,173.177,32.290,155.956
C06914=1063.166,247.497,409.165,173.180,32.293,155.956
C06915=1063.172,247.745,409.136,173.182,32.298,155.957
C06916=1063.177,247.993,409.108,173.185,32.301,155.958
C06917=1063.184,248.242,409.081,173.187,32.305,155.959
C06918=1063.189,248.490,409.053,173.188,32.309,155.959
C06919=1063.196,248.793,409.018,173.191,32.314,155.960
C06920=1063.204,249.095,408.984,173.194,32.319,155.961
C06921=1063.211,249.398,408.949,173.197,32.323,155.962
C06922=1063.218,249.701,408.914,173.200,32.328,155.963
C06923=1063.224,249.950,408.886,173.203,32.333,155.964
C06924=1063.231,250.198,408.858,173.205,32.336,155.964
C06925=1063.236,250.446,408.830,173.208,32.341,155.965
C06926=1063.242,250.695,408.802,173.210,32.344,155.966
C06927=1063.248,250.943,408.773,173.213,32.349,155.967
C06928=1063.254,251.192,408.745,173.214,32.352,155.967
C06929=1063.260,251.439,408.717,173.217,32.356,155.968
C06930=1063.266,251.688,408.689,173.219,32.360,155.969
C06931=1063.272,251.936,408.660,173.222,32.364,155.969
C06932=1063.278,252.185,408.632,173.224,32.368,155.970
C06933=1063.284,252.433,408.604,173.227,32.372,155.971
C06934=1063.291,252.681,408.575,173.229,32.376,155.972
C06935=1063.297,252.930,408.547,173.232,32.380,155.972
C06936=1063.303,253.178,408.519,173.234,32.384,155.973
C06937=1063.308,253.426,408.490,173.237,32.388,155.974
C06938=1063.314,253.675,408.462,173.239,32.392,155.975
C06939=1063.320,253.923,408.433,173.242,32.395,155.975
C06940=1063.327,254.171,408.405,173.244,32.400,155.976
C06941=1063.333,254.420,408.377,173.246,32.403,155.977
C06942=1063.339,254.667,408.348,173.248,32.407,155.977
C06943=1063.345,254.916,408.320,173.251,32.411,155.978
C06944=1063.351,255.164,408.291,173.253,32.415,155.979
C06945=1063.357,255.413,408.262,173.256,32.419,155.980
C06946=1063.364,255.661,408.234,173.258,32.423,155.980
C06947=1063.370,255.910,408.205,173.261,32.427,155.981
C06948=1063.376,256.158,408.176,173.263,32.431,155.982
C06949=1063.381,256.406,408.148,173.266,32.435,155.983
C06950=1063.388,256.654,408.119,173.268,32.438,155.983
C06951=1063.394,256.903,408.091,173.271,32.443,155.984
C06952=1063.400,257.151,408.062,173.274,32.446,155.985
C06953=1063.406,257.399,408.033,173.276,32.450,155.985
C06954=1063.413,257.647,408.005,173.279,32.454,155.986
C06955=1063.419,257.895,407.976,173.280,32.458,155.987
C06956=1063.425,258.144,407.948,173.283,32.462,155.988
C06957=1063.431,258.392,407.919,173.285,32.466,155.988
C06958=1063.437,258.640,407.890,173.288,32.470,155.989
C06959=1063.443,258.889,407.862,173.290,32.473,155.990
C06960=1063.450,259.137,407.832,173.293,32.478,155.990
C06961=1063.456,259.386,407.803,173.296,32.481,155.991
C06962=1063.461,259.634,407.775,173.298,32.485,155.992
C06963=1063.471,260.022,407.730,173.302,32.491,155.993
C06964=1063.481,260.411,407.686,173.306,32.497,155.994
C06965=1063.491,260.799,407.640,173.310,32.504,155.995
C06966=1063.501,261.188,407.595,173.314,32.510,155.996
C06967=1063.507,261.436,407.566,173.317,32.513,155.997
C06968=1063.513,261.684,407.537,173.319,32.517,155.998
C06969=1063.519,261.933,407.509,173.321,32.521,155.998
C06970=1063.525,262.181,407.480,173.324,32.525,155.999
C06971=1063.532,262.401,407.454,173.326,32.528,156.000
C06972=1063.537,262.622,407.428,173.328,32.532,156.000
C06973=1063.542,262.842,407.403,173.331,32.535,156.001
C06974=1063.548,263.063,407.377,173.333,32.539,156.002
C06975=1063.553,263.284,407.351,173.335,32.542,156.002
C06976=1063.560,263.504,407.325,173.338,32.545,156.003
C06977=1063.565,263.724,407.299,173.340,32.549,156.004
C06978=1063.570,263.945,407.273,173.342,32.553,156.004
C06979=1063.576,264.193,407.244,173.345,32.556,156.005
C06980=1063.582,264.442,407.215,173.347,32.561,156.006
C06981=1063.588,264.690,407.186,173.350,32.564,156.007
C06982=1063.594,264.938,407.157,173.353,32.568,156.007
C06983=1063.600,265.186,407.128,173.355,32.572,156.008
C06984=1063.606,265.434,407.098,173.358,32.576,156.009
C06985=1063.613,265.682,407.069,173.361,32.580,156.009
C06986=1063.618,265.930,407.039,173.362,32.584,156.010
C06987=1063.625,266.179,407.010,173.365,32.588,156.011
C06988=1063.631,266.427,406.981,173.367,32.592,156.012
C06989=1063.637,266.675,406.952,173.370,32.596,156.012
C06990=1063.643,266.923,406.922,173.373,32.600,156.013
C06991=1063.649,267.171,406.893,173.375,32.604,156.014
C06992=1063.655,267.419,406.864,173.378,32.608,156.015
C06993=1063.661,267.669,406.834,173.381,32.612,156.015
C06994=1063.668,267.916,406.804,173.383,32.616,156.016
C06995=1063.674,268.164,406.775,173.386,32.620,156.017
C06996=1063.680,268.413,406.746,173.389,32.623,156.017
C06997=1063.686,268.661,406.717,173.391,32.627,156.018
C06998=1063.692,268.909,406.688,173.394,32.631,156.019
C06999=1063.698,269.157,406.657,173.397,32.635,156.020
C07000=1063.704,269.405,406.628,173.399,32.639,156.020
C07001=1063.710,269.653,406.599,173.402,32.643,156.021
C07002=1063.717,269.902,406.569,173.405,32.647,156.022
C07003=1063.723,270.150,406.540,173.407,32.651,156.023
C07004=1063.729,270.398,406.510,173.410,32.655,156.023
C07005=1063.735,270.646,406.480,173.413,32.659,156.024
C07006=1063.741,270.894,406.451,173.415,32.663,156.025
C07007=1063.747,271.142,406.421,173.418,32.667,156.026
C07008=1063.753,271.391,406.391,173.420,32.671,156.026
C07009=1063.760,271.639,406.362,173.422,32.675,156.027
C07010=1063.765,271.887,406.332,173.425,32.679,156.028
C07011=1063.772,272.135,406.302,173.428,32.683,156.029
C07012=1063.778,272.383,406.273,173.430,32.687,156.029
C07013=1063.784,272.631,406.243,173.433,32.690,156.030
C07014=1063.791,272.880,406.214,173.436,32.695,156.031
C07015=1063.796,273.127,406.183,173.438,32.698,156.032
C07016=1063.802,273.376,406.154,173.441,32.703,156.032
C07017=1063.808,273.623,406.124,173.444,32.706,156.033
C07018=1063.814,273.872,406.094,173.446,32.711,156.034
C07019=1063.821,274.120,406.064,173.449,32.714,156.035
C07020=1063.827,274.369,406.034,173.452,32.719,156.035
C07021=1063.832,274.616,406.004,173.455,32.722,156.036
C07022=1063.839,274.864,405.974,173.457,32.726,156.037
C07023=1063.845,275.113,405.944,173.460,32.730,156.038
C07024=1063.851,275.361,405.914,173.463,32.734,156.038
C07025=1063.857,275.609,405.885,173.465,32.738,156.039
C07026=1063.863,275.857,405.855,173.468,32.742,156.040
C07027=1063.869,276.080,405.828,173.471,32.746,156.040
C07028=1063.874,276.301,405.801,173.473,32.749,156.041
C07029=1063.880,276.524,405.774,173.475,32.753,156.042
C07030=1063.886,276.746,405.747,173.478,32.756,156.042
C07031=1063.890,276.969,405.720,173.480,32.760,156.043
C07032=1063.896,277.191,405.693,173.483,32.764,156.044
C07033=1063.902,277.413,405.666,173.485,32.767,156.045
C07034=1063.907,277.635,405.639,173.488,32.771,156.045
C07035=1063.913,277.884,405.609,173.490,32.775,156.046
C07036=1063.919,278.132,405.579,173.493,32.779,156.047
C07037=1063.926,278.379,405.549,173.496,32.783,156.047
C07038=1063.932,278.628,405.518,173.499,32.787,156.048
C07039=1063.938,278.876,405.488,173.501,32.791,156.049
C07040=1063.944,279.124,405.459,173.503,32.795,156.050
C07041=1063.950,279.372,405.428,173.506,32.799,156.050
C07042=1063.956,279.620,405.398,173.509,32.803,156.051
C07043=1063.962,279.868,405.367,173.512,32.806,156.052
C07044=1063.969,280.116,405.337,173.514,32.811,156.053
C07045=1063.975,280.364,405.307,173.517,32.814,156.053
C07046=1063.981,280.613,405.276,173.520,32.819,156.054
C07047=1063.987,280.860,405.246,173.523,32.823,156.055
C07048=1063.993,281.108,405.216,173.525,32.826,156.056
C07049=1064.000,281.357,405.185,173.528,32.831,156.056
C07050=1064.005,281.605,405.154,173.531,32.835,156.057
C07051=1064.011,281.852,405.124,173.534,32.839,156.058
C07052=1064.018,282.101,405.093,173.536,32.843,156.059
C07053=1064.023,282.349,405.063,173.539,32.847,156.060
C07054=1064.029,282.597,405.033,173.542,32.851,156.060
C07055=1064.036,282.845,405.002,173.545,32.855,156.061
C07056=1064.041,283.093,404.972,173.548,32.859,156.062
C07057=1064.048,283.341,404.941,173.550,32.863,156.063
C07058=1064.054,283.589,404.911,173.553,32.867,156.063
C07059=1064.060,283.837,404.880,173.556,32.871,156.064
C07060=1064.067,284.085,404.850,173.559,32.875,156.065
C07061=1064.073,284.332,404.819,173.562,32.879,156.066
C07062=1064.079,284.581,404.788,173.564,32.883,156.066
C07063=1064.085,284.829,404.758,173.567,32.887,156.067
C07064=1064.091,285.077,404.727,173.570,32.892,156.068
C07065=1064.097,285.325,404.697,173.573,32.895,156.069
C07066=1064.104,285.573,404.665,173.576,32.900,156.069
C07067=1064.110,285.821,404.635,173.579,32.903,156.070
C07068=1064.116,286.069,404.605,173.581,32.907,156.071
C07069=1064.122,286.317,404.574,173.584,32.912,156.072
C07070=1064.129,286.565,404.543,173.587,32.915,156.072
C07071=1064.135,286.813,404.512,173.590,32.920,156.073
C07072=1064.141,287.061,404.482,173.593,32.924,156.074
C07073=1064.147,287.309,404.450,173.596,32.928,156.075
C07074=1064.154,287.557,404.420,173.598,32.932,156.076
C07075=1064.159,287.805,404.389,173.601,32.936,156.076
C07076=1064.165,288.053,404.357,173.604,32.940,156.077
C07077=1064.171,288.301,404.327,173.607,32.944,156.078
C07078=1064.178,288.550,404.296,173.610,32.948,156.079
C07079=1064.184,288.797,404.265,173.613,32.952,156.079
C07080=1064.190,289.045,404.235,173.616,32.956,156.080
C07081=1064.196,289.292,404.203,173.618,32.960,156.081
C07082=1064.203,289.541,404.173,173.621,32.964,156.082
C07083=1064.208,289.768,404.143,173.624,32.968,156.083
C07084=1064.214,289.996,404.115,173.627,32.972,156.083
C07085=1064.219,290.223,404.087,173.629,32.975,156.084
C07086=1064.225,290.451,404.058,173.632,32.979,156.085
C07087=1064.231,290.679,404.030,173.635,32.983,156.085
C07088=1064.237,290.907,404.002,173.637,32.987,156.086
C07089=1064.242,291.134,403.972,173.640,32.991,156.087
C07090=1064.248,291.362,403.944,173.642,32.994,156.088
C07091=1064.254,291.609,403.913,173.645,32.998,156.088
C07092=1064.260,291.858,403.882,173.648,33.003,156.089
C07093=1064.266,292.105,403.851,173.651,33.006,156.090
C07094=1064.272,292.353,403.819,173.654,33.011,156.091
C07095=1064.279,292.602,403.788,173.657,33.015,156.091
C07096=1064.285,292.849,403.757,173.660,33.019,156.092
C07097=1064.291,293.097,403.725,173.663,33.023,156.093
C07098=1064.297,293.346,403.694,173.666,33.027,156.094
C07099=1064.303,293.593,403.663,173.669,33.031,156.095
C07100=1064.310,293.841,403.632,173.671,33.035,156.095
C07101=1064.316,294.089,403.600,173.674,33.040,156.096
C07102=1064.322,294.337,403.569,173.677,33.043,156.097
C07103=1064.329,294.585,403.538,173.680,33.047,156.098
C07104=1064.335,294.833,403.506,173.683,33.052,156.099
C07105=1064.341,295.080,403.475,173.686,33.056,156.099
C07106=1064.347,295.328,403.443,173.689,33.060,156.100
C07107=1064.353,295.577,403.412,173.692,33.064,156.101
C07108=1064.359,295.824,403.381,173.695,33.068,156.102
C07109=1064.365,296.072,403.349,173.698,33.072,156.102
C07110=1064.372,296.320,403.318,173.701,33.077,156.103
C07111=1064.377,296.568,403.286,173.704,33.081,156.104
C07112=1064.384,296.816,403.255,173.707,33.085,156.105
C07113=1064.390,297.064,403.223,173.710,33.089,156.106
C07114=1064.397,297.312,403.191,173.713,33.093,156.107
C07115=1064.402,297.559,403.159,173.715,33.098,156.107
C07116=1064.408,297.807,403.127,173.718,33.102,156.108
C07117=1064.415,298.055,403.096,173.721,33.106,156.109
C07118=1064.420,298.303,403.064,173.724,33.110,156.110
C07119=1064.426,298.551,403.032,173.727,33.114,156.111
C07120=1064.433,298.799,403.001,173.730,33.119,156.111
C07121=1064.438,299.046,402.969,173.734,33.123,156.112
C07122=1064.444,299.295,402.937,173.737,33.127,156.113
C07123=1064.451,299.542,402.904,173.740,33.131,156.114
C07124=1064.457,299.790,402.873,173.743,33.136,156.115
C07125=1064.463,300.038,402.841,173.746,33.140,156.116
C07126=1064.469,300.286,402.809,173.749,33.144,156.116
C07127=1064.475,300.534,402.777,173.752,33.148,156.117
C07128=1064.481,300.782,402.746,173.755,33.152,156.118
C07129=1064.487,301.029,402.713,173.758,33.157,156.119
C07130=1064.493,301.277,402.681,173.761,33.161,156.120
C07131=1064.499,301.525,402.649,173.764,33.166,156.121
C07132=1064.506,301.773,402.617,173.767,33.170,156.121
C07133=1064.512,302.021,402.585,173.770,33.174,156.122
C07134=1064.517,302.268,402.554,173.773,33.178,156.123
C07135=1064.523,302.517,402.522,173.776,33.182,156.124
C07136=1064.530,302.764,402.489,173.779,33.187,156.125
C07137=1064.536,303.012,402.457,173.782,33.191,156.125
C07138=1064.542,303.260,402.425,173.785,33.195,156.126
C07139=1064.549,303.495,402.394,173.788,33.199,156.127
C07140=1064.554,303.730,402.364,173.791,33.204,156.128
C07141=1064.560,303.965,402.333,173.794,33.207,156.129
C07142=1064.566,304.200,402.303,173.796,33.211,156.129
C07143=1064.572,304.435,402.273,173.799,33.215,156.130
C07144=1064.578,304.670,402.242,173.802,33.220,156.131
C07145=1064.584,304.906,402.212,173.805,33.223,156.132
C07146=1064.590,305.141,402.181,173.808,33.228,156.133
C07147=1064.596,305.388,402.149,173.811,33.232,156.133
C07148=1064.602,305.636,402.117,173.814,33.236,156.134
C07149=1064.608,305.884,402.084,173.818,33.240,156.135
C07150=1064.614,306.132,402.052,173.821,33.245,156.136
C07151=1064.621,306.380,402.020,173.824,33.249,156.137
C07152=1064.627,306.627,401.987,173.827,33.253,156.138
C07153=1064.633,306.875,401.955,173.830,33.258,156.138
C07154=1064.640,307.123,401.922,173.834,33.262,156.139
C07155=1064.646,307.371,401.890,173.837,33.266,156.140
C07156=1064.652,307.619,401.858,173.840,33.270,156.141
C07157=1064.659,307.866,401.825,173.843,33.275,156.142
C07158=1064.665,308.114,401.793,173.846,33.279,156.143
C07159=1064.671,308.362,401.761,173.849,33.283,156.143
C07160=1064.678,308.609,401.728,173.852,33.288,156.144
C07161=1064.684,308.858,401.696,173.855,33.292,156.145
C07162=1064.690,309.105,401.663,173.858,33.296,156.146
C07163=1064.696,309.353,401.630,173.861,33.300,156.147
C07164=1064.702,309.600,401.598,173.864,33.305,156.148
C07165=1064.709,309.848,401.566,173.868,33.309,156.148
C07166=1064.715,310.096,401.533,173.871,33.313,156.149
C07167=1064.722,310.344,401.501,173.874,33.318,156.150
C07168=1064.729,310.592,401.468,173.877,33.322,156.151
C07169=1064.735,310.839,401.435,173.881,33.327,156.152
C07170=1064.741,311.088,401.403,173.884,33.331,156.153
C07171=1064.747,311.335,401.370,173.887,33.335,156.154
C07172=1064.754,311.583,401.337,173.890,33.339,156.154
C07173=1064.760,311.830,401.305,173.894,33.343,156.155
C07174=1064.766,312.078,401.272,173.897,33.348,156.156
C07175=1064.773,312.326,401.239,173.900,33.352,156.157
C07176=1064.780,312.574,401.207,173.903,33.356,156.158
C07177=1064.786,312.821,401.174,173.906,33.361,156.159
C07178=1064.793,313.069,401.141,173.909,33.365,156.159
C07179=1064.799,313.316,401.108,173.912,33.370,156.160
C07180=1064.806,313.565,401.075,173.916,33.374,156.161
C07181=1064.812,313.812,401.042,173.919,33.378,156.162
C07182=1064.818,314.060,401.010,173.922,33.382,156.163
C07183=1064.824,314.308,400.976,173.925,33.387,156.164
C07184=1064.830,314.555,400.944,173.929,33.391,156.165
C07185=1064.836,314.804,400.910,173.932,33.396,156.166
C07186=1064.843,315.052,400.877,173.935,33.401,156.166
C07187=1064.849,315.299,400.844,173.939,33.405,156.167
C07188=1064.855,315.546,400.810,173.942,33.410,156.168
C07189=1064.861,315.794,400.778,173.945,33.414,156.169
C07190=1064.867,316.042,400.744,173.948,33.419,156.170
C07191=1064.873,316.289,400.712,173.951,33.423,156.171
C07192=1064.880,316.537,400.678,173.954,33.427,156.172
C07193=1064.886,316.785,400.644,173.957,33.432,156.173
C07194=1064.892,317.033,400.612,173.961,33.436,156.174
C07195=1064.898,317.270,400.579,173.964,33.441,156.174
C07196=1064.904,317.507,400.548,173.967,33.445,156.175
C07197=1064.909,317.744,400.515,173.971,33.449,156.176
C07198=1064.916,317.981,400.484,173.974,33.454,156.177
C07199=1064.922,318.218,400.452,173.977,33.458,156.178
C07200=1064.928,318.455,400.420,173.980,33.463,156.179
C07201=1064.934,318.692,400.388,173.983,33.467,156.180
C07202=1064.939,318.928,400.356,173.986,33.471,156.181
C07203=1064.946,319.176,400.323,173.989,33.476,156.181
C07204=1064.952,319.424,400.289,173.992,33.480,156.182
C07205=1064.958,319.671,400.256,173.996,33.485,156.183
C07206=1064.964,319.919,400.222,173.999,33.489,156.184
C07207=1064.971,320.167,400.189,174.002,33.494,156.185
C07208=1064.977,320.414,400.155,174.006,33.498,156.186
C07209=1064.983,320.662,400.122,174.009,33.503,156.187
C07210=1064.989,320.910,400.088,174.013,33.508,156.188
C07211=1064.996,321.157,400.055,174.016,33.512,156.189
C07212=1065.002,321.405,400.020,174.019,33.517,156.190
C07213=1065.008,321.653,399.988,174.022,33.521,156.190
C07214=1065.014,321.900,399.954,174.026,33.526,156.191
C07215=1065.021,322.148,399.920,174.029,33.530,156.192
C07216=1065.027,322.396,399.887,174.032,33.535,156.193
C07217=1065.034,322.643,399.853,174.035,33.540,156.194
C07218=1065.040,322.891,399.819,174.040,33.544,156.195
C07219=1065.046,323.139,399.785,174.043,33.549,156.196
C07220=1065.053,323.386,399.751,174.046,33.553,156.197
C07221=1065.059,323.634,399.717,174.049,33.558,156.198
C07222=1065.066,323.882,399.684,174.053,33.562,156.199
C07223=1065.071,324.129,399.650,174.056,33.567,156.200
C07224=1065.079,324.377,399.616,174.059,33.572,156.201
C07225=1065.084,324.624,399.582,174.062,33.576,156.202
C07226=1065.091,324.872,399.549,174.066,33.581,156.202
C07227=1065.097,325.120,399.515,174.069,33.585,156.203
C07228=1065.104,325.368,399.481,174.073,33.590,156.204
C07229=1065.110,325.615,399.447,174.077,33.595,156.205
C07230=1065.117,325.863,399.413,174.080,33.599,156.206
C07231=1065.124,326.110,399.379,174.083,33.604,156.207
C07232=1065.130,326.358,399.345,174.086,33.608,156.208
C07233=1065.136,326.606,399.311,174.090,33.613,156.209
C07234=1065.143,326.853,399.278,174.093,33.618,156.210
C07235=1065.149,327.101,399.243,174.096,33.623,156.211
C07236=1065.156,327.348,399.210,174.101,33.627,156.212
C07237=1065.162,327.596,399.176,174.104,33.632,156.213
C07238=1065.169,327.844,399.141,174.107,33.637,156.214
C07239=1065.175,328.091,399.108,174.111,33.641,156.214
C07240=1065.182,328.339,399.073,174.114,33.646,156.215
C07241=1065.188,328.587,399.039,174.117,33.650,156.216
C07242=1065.195,328.833,399.005,174.121,33.655,156.217
C07243=1065.201,329.081,398.970,174.124,33.660,156.218
C07244=1065.208,329.329,398.936,174.128,33.664,156.219
C07245=1065.214,329.576,398.902,174.132,33.669,156.220
C07246=1065.221,329.824,398.868,174.135,33.674,156.221
C07247=1065.227,330.072,398.834,174.139,33.679,156.222
C07248=1065.234,330.319,398.800,174.142,33.683,156.223
C07249=1065.240,330.567,398.766,174.145,33.688,156.224
C07250=1065.247,330.815,398.731,174.149,33.693,156.225
C07251=1065.254,331.049,398.699,174.152,33.697,156.226
C07252=1065.259,331.283,398.666,174.156,33.702,156.227
C07253=1065.265,331.516,398.633,174.159,33.706,156.228
C07254=1065.271,331.751,398.601,174.162,33.711,156.229
C07255=1065.277,331.985,398.568,174.166,33.715,156.230
C07256=1065.284,332.219,398.535,174.169,33.720,156.230
C07257=1065.289,332.453,398.502,174.172,33.725,156.231
C07258=1065.295,332.687,398.470,174.175,33.729,156.232
C07259=1065.302,332.935,398.435,174.179,33.734,156.233
C07260=1065.308,333.182,398.401,174.183,33.739,156.234
C07261=1065.314,333.429,398.366,174.186,33.744,156.235
C07262=1065.321,333.677,398.331,174.190,33.749,156.236
C07263=1065.328,333.925,398.296,174.193,33.753,156.237
C07264=1065.333,334.172,398.262,174.196,33.758,156.238
C07265=1065.340,334.419,398.227,174.200,33.763,156.239
C07266=1065.347,334.667,398.193,174.204,33.768,156.240
C07267=1065.353,334.915,398.157,174.208,33.773,156.241
C07268=1065.359,335.162,398.123,174.211,33.778,156.242
C07269=1065.366,335.409,398.088,174.215,33.783,156.243
C07270=1065.373,335.657,398.054,174.218,33.787,156.244
C07271=1065.379,335.905,398.019,174.221,33.793,156.245
C07272=1065.386,336.152,397.984,174.225,33.797,156.246
C07273=1065.393,336.400,397.949,174.229,33.802,156.247
C07274=1065.399,336.647,397.914,174.233,33.807,156.248
C07275=1065.405,336.894,397.879,174.236,33.812,156.249
C07276=1065.411,337.142,397.844,174.240,33.817,156.250
C07277=1065.418,337.390,397.809,174.243,33.822,156.251
C07278=1065.425,337.637,397.774,174.247,33.827,156.252
C07279=1065.431,337.884,397.739,174.251,33.832,156.253
C07280=1065.437,338.133,397.704,174.254,33.837,156.254
C07281=1065.443,338.379,397.669,174.258,33.842,156.255
C07282=1065.450,338.627,397.634,174.261,33.847,156.257
C07283=1065.457,338.874,397.599,174.265,33.852,156.257
C07284=1065.463,339.122,397.563,174.269,33.857,156.259
C07285=1065.470,339.369,397.528,174.273,33.862,156.260
